LIN {X 0,Y 411.208,Z 237.264,A -85,B 0,C 180,E1 -10473.156,E2 -10473.156} C_VEL
LIN {X 0,Y 411.193,Z 237.263,A -85,B 0,C 180,E1 -10476.552,E2 -10476.552} C_VEL
LIN {X 0,Y 411.171,Z 237.27,A -85,B 0,C 180,E1 -10479.72,E2 -10479.72} C_VEL
LIN {X 0,Y 411.166,Z 237.272,A -85,B 0,C 180,E1 -10483.135,E2 -10483.135} C_VEL
LIN {X 0,Y 411.208,Z 237.375,A -85,B 0,C 180,E1 -10486.787,E2 -10486.787} C_VEL
LIN {X 0,Y 412.368,Z 243.528,A -85,B 0,C 180,E1 -10490.08,E2 -10490.08} C_VEL
LIN {X 0,Y 413.369,Z 249.555,A -85,B 0,C 180,E1 -10493.043,E2 -10493.043} C_VEL
LIN {X 0,Y 413.313,Z 254.436,A -85,B 0,C 180,E1 -10495.275,E2 -10495.275} C_VEL
LIN {X 0,Y 412.67,Z 262.638,A -85,B 0,C 180,E1 -10498.816,E2 -10498.816} C_VEL
LIN {X 0,Y 412.048,Z 271.447,A -85,B 0,C 180,E1 -10502.49,E2 -10502.49} C_VEL
LIN {X 0,Y 411.535,Z 279.596,A -85,B 0,C 180,E1 -10505.804,E2 -10505.804} C_VEL
LIN {X 0,Y 411.103,Z 287.435,A -85,B 0,C 180,E1 -10508.961,E2 -10508.961} C_VEL
LIN {X 0,Y 410.706,Z 295.977,A -85,B 0,C 180,E1 -10512.395,E2 -10512.395} C_VEL
LIN {X 0,Y 413.028,Z 310.701,A -85,B 0,C 180,E1 -10512.959,E2 -10512.959} C_VEL
LIN {X 0,Y 414.855,Z 323.572,A -85,B 0,C 180,E1 -10513.644,E2 -10513.644} C_VEL
LIN {X 0,Y 414.255,Z 335.281,A -85,B 0,C 180,E1 -10514.376,E2 -10514.376} C_VEL
LIN {X 0,Y 413.474,Z 345.991,A -85,B 0,C 180,E1 -10515.229,E2 -10515.229} C_VEL
LIN {X 0,Y 412.699,Z 356.944,A -85,B 0,C 180,E1 -10516.333,E2 -10516.333} C_VEL
LIN {X 0,Y 412.139,Z 365.888,A -85,B 0,C 180,E1 -10517.443,E2 -10517.443} C_VEL
LIN {X 0,Y 411.369,Z 375.605,A -85,B 0,C 180,E1 -10518.919,E2 -10518.919} C_VEL
LIN {X 0,Y 410.826,Z 383.351,A -85,B 0,C 180,E1 -10520.399,E2 -10520.399} C_VEL
LIN {X 0,Y 410.354,Z 390.497,A -85,B 0,C 180,E1 -10522.125,E2 -10522.125} C_VEL
LIN {X 0,Y 410.177,Z 395.261,A -85,B 0,C 180,E1 -10523.606,E2 -10523.606} C_VEL
LIN {X 0,Y 410.096,Z 398.905,A -85,B 0,C 180,E1 -10525.085,E2 -10525.085} C_VEL
LIN {X 0,Y 409.954,Z 400.778,A -85,B 0,C 180,E1 -10526.068,E2 -10526.068} C_VEL
LIN {X 0,Y 410.007,Z 402.193,A -85,B 0,C 180,E1 -10527.052,E2 -10527.052} C_VEL
LIN {X 0,Y 409.988,Z 403.2,A -85,B 0,C 180,E1 -10528.035,E2 -10528.035} C_VEL
LIN {X 0,Y 409.959,Z 403.813,A -85,B 0,C 180,E1 -10529.018,E2 -10529.018} C_VEL
LIN {X 0,Y 409.967,Z 404.032,A -85,B 0,C 180,E1 -10530,E2 -10530} C_VEL
LIN {X 0,Y 409.959,Z 403.813,A -85,B 0,C 180,E1 -10530.982,E2 -10530.982} C_VEL
LIN {X 0,Y 409.988,Z 403.201,A -85,B 0,C 180,E1 -10531.965,E2 -10531.965} C_VEL
LIN {X 0,Y 410.007,Z 402.196,A -85,B 0,C 180,E1 -10532.948,E2 -10532.948} C_VEL
LIN {X 0,Y 409.954,Z 400.782,A -85,B 0,C 180,E1 -10533.932,E2 -10533.932} C_VEL
LIN {X 0,Y 410.108,Z 397.823,A -85,B 0,C 180,E1 -10535.409,E2 -10535.409} C_VEL
LIN {X 0,Y 410.198,Z 393.812,A -85,B 0,C 180,E1 -10536.888,E2 -10536.888} C_VEL
LIN {X 0,Y 410.551,Z 387.657,A -85,B 0,C 180,E1 -10538.615,E2 -10538.615} C_VEL
LIN {X 0,Y 410.993,Z 380.936,A -85,B 0,C 180,E1 -10540.095,E2 -10540.095} C_VEL
LIN {X 0,Y 411.602,Z 372.606,A -85,B 0,C 180,E1 -10541.574,E2 -10541.574} C_VEL
LIN {X 0,Y 412.221,Z 364.073,A -85,B 0,C 180,E1 -10542.806,E2 -10542.806} C_VEL
LIN {X 0,Y 412.945,Z 354.501,A -85,B 0,C 180,E1 -10543.934,E2 -10543.934} C_VEL
LIN {X 0,Y 413.672,Z 343.125,A -85,B 0,C 180,E1 -10545.016,E2 -10545.016} C_VEL
LIN {X 0,Y 414.506,Z 331.727,A -85,B 0,C 180,E1 -10545.867,E2 -10545.867} C_VEL
LIN {X 0,Y 414.812,Z 323.512,A -85,B 0,C 180,E1 -10546.36,E2 -10546.36} C_VEL
LIN {X 0,Y 412.966,Z 310.197,A -85,B 0,C 180,E1 -10547.063,E2 -10547.063} C_VEL
LIN {X 0,Y 410.827,Z 297.222,A -85,B 0,C 180,E1 -10547.554,E2 -10547.554} C_VEL
LIN {X 0,Y 410.719,Z 295.854,A -85,B 0,C 180,E1 -10547.636,E2 -10547.636} C_VEL
LIN {X 0,Y 411.108,Z 287.427,A -85,B 0,C 180,E1 -10551.039,E2 -10551.039} C_VEL
LIN {X 0,Y 411.529,Z 279.586,A -85,B 0,C 180,E1 -10554.197,E2 -10554.197} C_VEL
LIN {X 0,Y 412.03,Z 271.406,A -85,B 0,C 180,E1 -10557.506,E2 -10557.506} C_VEL
LIN {X 0,Y 412.548,Z 263.641,A -85,B 0,C 180,E1 -10560.735,E2 -10560.735} C_VEL
LIN {X 0,Y 413.078,Z 257.152,A -85,B 0,C 180,E1 -10563.522,E2 -10563.522} C_VEL
LIN {X 0,Y 413.457,Z 251.781,A -85,B 0,C 180,E1 -10565.905,E2 -10565.905} C_VEL
LIN {X 0,Y 413.12,Z 247.857,A -85,B 0,C 180,E1 -10567.766,E2 -10567.766} C_VEL
LIN {X 0,Y 411.88,Z 240.822,A -85,B 0,C 180,E1 -10571.342,E2 -10571.342} C_VEL
LIN {X 0,Y 411.202,Z 237.271,A -85,B 0,C 180,E1 -10573.298,E2 -10573.298} C_VEL
LIN {X 0,Y 411.167,Z 237.271,A -85,B 0,C 180,E1 -10576.865,E2 -10576.865} C_VEL
LIN {X 0,Y 411.172,Z 237.267,A -85,B 0,C 180,E1 -10580.28,E2 -10580.28} C_VEL
LIN {X 0,Y 411.195,Z 237.263,A -85,B 0,C 180,E1 -10583.448,E2 -10583.448} C_VEL
LIN {X 0,Y 411.211,Z 237.264,A -85,B 0,C 180,E1 -10586.874,E2 -10586.874} C_VEL
LIN {X 0,Y 411.214,Z 237.264,A -85,B 0,C 180,E1 -10590.65,E2 -10590.65} C_VEL
LIN {X 0,Y 411.179,Z 237.264,A -85,B 0,C 180,E1 -10593.615,E2 -10593.615} C_VEL
LIN {X 0,Y 411.193,Z 237.263,A -85,B 0,C 180,E1 -10596.852,E2 -10596.852} C_VEL
LIN {X 0,Y 411.219,Z 237.264,A -85,B 0,C 180,E1 -10600.05,E2 -10600.05} C_VEL
LIN {X 0,Y 411.267,Z 237.254,A -85,B 0,C 180,E1 -10603.131,E2 -10603.131} C_VEL
LIN {X 0,Y 411.309,Z 237.248,A -85,B 0,C 180,E1 -10606.897,E2 -10606.897} C_VEL
LIN {X 0,Y 411.282,Z 237.254,A -85,B 0,C 180,E1 -10610.161,E2 -10610.161} C_VEL
LIN {X 0,Y 411.442,Z 237.233,A -85,B 0,C 180,E1 -10613.133,E2 -10613.133} C_VEL
LIN {X 0,Y 411.312,Z 237.25,A -85,B 0,C 180,E1 -10615.099,E2 -10615.099} C_VEL
LIN {X 0,Y 411.515,Z 237.224,A -85,B 0,C 180,E1 -10618.043,E2 -10618.043} C_VEL
LIN {X 0,Y 411.382,Z 237.241,A -85,B 0,C 180,E1 -10620.979,E2 -10620.979} C_VEL
LIN {X 0,Y 411.443,Z 237.233,A -85,B 0,C 180,E1 -10622.937,E2 -10622.937} C_VEL
LIN {X 0,Y 411.437,Z 237.233,A -85,B 0,C 180,E1 -10626.648,E2 -10626.648} C_VEL
LIN {X 0,Y 411.324,Z 237.25,A -85,B 0,C 180,E1 -10628.846,E2 -10628.846} C_VEL
LIN {X 0,Y 411.289,Z 237.252,A -85,B 0,C 180,E1 -10631.833,E2 -10631.833} C_VEL
LIN {X 0,Y 411.256,Z 237.258,A -85,B 0,C 180,E1 -10634.853,E2 -10634.853} C_VEL
LIN {X 0,Y 411.248,Z 237.255,A -85,B 0,C 180,E1 -10637.915,E2 -10637.915} C_VEL
LIN {X 0,Y 411.201,Z 237.265,A -85,B 0,C 180,E1 -10641.034,E2 -10641.034} C_VEL
LIN {X 0,Y 411.216,Z 237.262,A -85,B 0,C 180,E1 -10644.216,E2 -10644.216} C_VEL
LIN {X 0,Y 411.183,Z 237.264,A -85,B 0,C 180,E1 -10647.483,E2 -10647.483} C_VEL
LIN {X 0,Y 411.199,Z 237.262,A -85,B 0,C 180,E1 -10649.713,E2 -10649.713} C_VEL
LIN {X 0,Y 411.21,Z 237.261,A -85,B 0,C 180,E1 -10653.156,E2 -10653.156} C_VEL
LIN {X 0,Y 411.196,Z 237.266,A -85,B 0,C 180,E1 -10656.552,E2 -10656.552} C_VEL
LIN {X 0,Y 411.21,Z 237.263,A -85,B 0,C 180,E1 -10659.727,E2 -10659.727} C_VEL
LIN {X 0,Y 411.174,Z 237.265,A -85,B 0,C 180,E1 -10663.134,E2 -10663.134} C_VEL
LIN {X 0,Y 411.171,Z 237.269,A -85,B 0,C 180,E1 -10665.881,E2 -10665.881} C_VEL
LIN {X 0,Y 411.163,Z 237.267,A -85,B 0,C 180,E1 -10668.772,E2 -10668.772} C_VEL
LIN {X 0,Y 411.191,Z 237.267,A -85,B 0,C 180,E1 -10672.025,E2 -10672.025} C_VEL
LIN {X 0,Y 411.078,Z 237.279,A -85,B 0,C 180,E1 -10675.149,E2 -10675.149} C_VEL
LIN {X 0,Y 410.719,Z 237.327,A -85,B 0,C 180,E1 -10677.963,E2 -10677.963} C_VEL
LIN {X 0,Y 410.617,Z 239.167,A -85,B 0,C 180,E1 -10680.24,E2 -10680.24} C_VEL
LIN {X 0,Y 410.512,Z 242.3,A -85,B 0,C 180,E1 -10683.569,E2 -10683.569} C_VEL
LIN {X 0,Y 410.497,Z 244.4,A -85,B 0,C 180,E1 -10685.738,E2 -10685.738} C_VEL
LIN {X 0,Y 410.419,Z 247.648,A -85,B 0,C 180,E1 -10688.924,E2 -10688.924} C_VEL
LIN {X 0,Y 410.4,Z 251.592,A -85,B 0,C 180,E1 -10692.501,E2 -10692.501} C_VEL
LIN {X 0,Y 414.208,Z 265.973,A -85,B 0,C 180,E1 -10693.18,E2 -10693.18} C_VEL
LIN {X 0,Y 415.689,Z 273.997,A -85,B 0,C 180,E1 -10693.638,E2 -10693.638} C_VEL
LIN {X 0,Y 415.064,Z 286.501,A -85,B 0,C 180,E1 -10694.407,E2 -10694.407} C_VEL
LIN {X 0,Y 414.427,Z 297.234,A -85,B 0,C 180,E1 -10695.263,E2 -10695.263} C_VEL
LIN {X 0,Y 413.779,Z 307.095,A -85,B 0,C 180,E1 -10696.244,E2 -10696.244} C_VEL
LIN {X 0,Y 412.992,Z 317.038,A -85,B 0,C 180,E1 -10697.469,E2 -10697.469} C_VEL
LIN {X 0,Y 412.244,Z 326.64,A -85,B 0,C 180,E1 -10698.942,E2 -10698.942} C_VEL
LIN {X 0,Y 411.583,Z 334.299,A -85,B 0,C 180,E1 -10700.416,E2 -10700.416} C_VEL
LIN {X 0,Y 411.025,Z 341.318,A -85,B 0,C 180,E1 -10702.138,E2 -10702.138} C_VEL
LIN {X 0,Y 410.699,Z 345.99,A -85,B 0,C 180,E1 -10703.614,E2 -10703.614} C_VEL
LIN {X 0,Y 410.418,Z 349.569,A -85,B 0,C 180,E1 -10705.088,E2 -10705.088} C_VEL
LIN {X 0,Y 410.412,Z 351.41,A -85,B 0,C 180,E1 -10706.072,E2 -10706.072} C_VEL
LIN {X 0,Y 410.276,Z 352.804,A -85,B 0,C 180,E1 -10707.054,E2 -10707.054} C_VEL
LIN {X 0,Y 410.078,Z 354.408,A -85,B 0,C 180,E1 -10709.018,E2 -10709.018} C_VEL
LIN {X 0,Y 410.074,Z 354.64,A -85,B 0,C 180,E1 -10710,E2 -10710} C_VEL
LIN {X 0,Y 410.139,Z 353.873,A -85,B 0,C 180,E1 -10711.964,E2 -10711.964} C_VEL
LIN {X 0,Y 410.408,Z 351.56,A -85,B 0,C 180,E1 -10713.928,E2 -10713.928} C_VEL
LIN {X 0,Y 410.42,Z 348.726,A -85,B 0,C 180,E1 -10715.404,E2 -10715.404} C_VEL
LIN {X 0,Y 410.796,Z 344.12,A -85,B 0,C 180,E1 -10717.123,E2 -10717.123} C_VEL
LIN {X 0,Y 411.267,Z 337.92,A -85,B 0,C 180,E1 -10718.847,E2 -10718.847} C_VEL
LIN {X 0,Y 411.417,Z 336.229,A -85,B 0,C 180,E1 -10719.249,E2 -10719.249} C_VEL
LIN {X 0,Y 411.057,Z 333.143,A -85,B 0,C 180,E1 -10719.946,E2 -10719.946} C_VEL
LIN {X 0,Y 407.66,Z 325.609,A -85,B 0,C 180,E1 -10721.511,E2 -10721.511} C_VEL
LIN {X 0,Y 406.164,Z 320.726,A -85,B 0,C 180,E1 -10722.362,E2 -10722.362} C_VEL
LIN {X 0,Y 406.065,Z 318.007,A -85,B 0,C 180,E1 -10722.768,E2 -10722.768} C_VEL
LIN {X 0,Y 406.893,Z 308.344,A -85,B 0,C 180,E1 -10723.994,E2 -10723.994} C_VEL
LIN {X 0,Y 407.587,Z 297.853,A -85,B 0,C 180,E1 -10725.07,E2 -10725.07} C_VEL
LIN {X 0,Y 408.319,Z 286.508,A -85,B 0,C 180,E1 -10725.985,E2 -10725.985} C_VEL
LIN {X 0,Y 408.902,Z 274.466,A -85,B 0,C 180,E1 -10726.737,E2 -10726.737} C_VEL
LIN {X 0,Y 406.265,Z 262.744,A -85,B 0,C 180,E1 -10727.417,E2 -10727.417} C_VEL
LIN {X 0,Y 403.333,Z 251.921,A -85,B 0,C 180,E1 -10727.934,E2 -10727.934} C_VEL
LIN {X 0,Y 403.334,Z 249.256,A -85,B 0,C 180,E1 -10730.395,E2 -10730.395} C_VEL
LIN {X 0,Y 403.403,Z 245.95,A -85,B 0,C 180,E1 -10733.622,E2 -10733.622} C_VEL
LIN {X 0,Y 403.481,Z 242.745,A -85,B 0,C 180,E1 -10736.929,E2 -10736.929} C_VEL
LIN {X 0,Y 403.612,Z 239.579,A -85,B 0,C 180,E1 -10740.329,E2 -10740.329} C_VEL
LIN {X 0,Y 403.631,Z 238.502,A -85,B 0,C 180,E1 -10741.491,E2 -10741.491} C_VEL
LIN {X 0,Y 403.873,Z 238.178,A -85,B 0,C 180,E1 -10743.838,E2 -10743.838} C_VEL
LIN {X 0,Y 404.097,Z 238.151,A -85,B 0,C 180,E1 -10746.251,E2 -10746.251} C_VEL
LIN {X 0,Y 404.15,Z 238.141,A -85,B 0,C 180,E1 -10748.758,E2 -10748.758} C_VEL
LIN {X 0,Y 404.121,Z 238.145,A -85,B 0,C 180,E1 -10751.599,E2 -10751.599} C_VEL
LIN {X 0,Y 404.147,Z 238.141,A -85,B 0,C 180,E1 -10754.522,E2 -10754.522} C_VEL
LIN {X 0,Y 404.134,Z 238.143,A -85,B 0,C 180,E1 -10757.295,E2 -10757.295} C_VEL
LIN {X 0,Y 404.171,Z 238.142,A -85,B 0,C 180,E1 -10759.955,E2 -10759.955} C_VEL
LIN {X 0,Y 404.137,Z 238.143,A -85,B 0,C 180,E1 -10763.125,E2 -10763.125} C_VEL
LIN {X 0,Y 404.147,Z 238.141,A -85,B 0,C 180,E1 -10766.188,E2 -10766.188} C_VEL
LIN {X 0,Y 404.146,Z 238.144,A -85,B 0,C 180,E1 -10769.715,E2 -10769.715} C_VEL
LIN {X 0,Y 404.131,Z 238.146,A -85,B 0,C 180,E1 -10773.118,E2 -10773.118} C_VEL
LIN {X 0,Y 404.163,Z 238.139,A -85,B 0,C 180,E1 -10776.425,E2 -10776.425} C_VEL
LIN {X 0,Y 404.194,Z 238.135,A -85,B 0,C 180,E1 -10779.874,E2 -10779.874} C_VEL
LIN {X 0,Y 404.218,Z 238.136,A -85,B 0,C 180,E1 -10782.993,E2 -10782.993} C_VEL
LIN {X 0,Y 404.285,Z 238.128,A -85,B 0,C 180,E1 -10786.939,E2 -10786.939} C_VEL
LIN {X 0,Y 404.261,Z 238.126,A -85,B 0,C 180,E1 -10789.988,E2 -10789.988} C_VEL
LIN {X 0,Y 404.413,Z 238.112,A -85,B 0,C 180,E1 -10793.013,E2 -10793.013} C_VEL
LIN {X 0,Y 404.277,Z 238.127,A -85,B 0,C 180,E1 -10795.013,E2 -10795.013} C_VEL
LIN {X 0,Y 404.477,Z 238.099,A -85,B 0,C 180,E1 -10798.008,E2 -10798.008} C_VEL
LIN {X 0,Y 404.412,Z 238.109,A -85,B 0,C 180,E1 -10800.996,E2 -10800.996} C_VEL
LIN {X 0,Y 404.418,Z 238.108,A -85,B 0,C 180,E1 -10802.988,E2 -10802.988} C_VEL
LIN {X 0,Y 404.417,Z 238.109,A -85,B 0,C 180,E1 -10805.985,E2 -10805.985} C_VEL
LIN {X 0,Y 404.265,Z 238.126,A -85,B 0,C 180,E1 -10809.002,E2 -10809.002} C_VEL
LIN {X 0,Y 404.252,Z 238.131,A -85,B 0,C 180,E1 -10812.042,E2 -10812.042} C_VEL
LIN {X 0,Y 404.207,Z 238.133,A -85,B 0,C 180,E1 -10815.118,E2 -10815.118} C_VEL
LIN {X 0,Y 404.213,Z 238.136,A -85,B 0,C 180,E1 -10818.238,E2 -10818.238} C_VEL
LIN {X 0,Y 404.141,Z 238.143,A -85,B 0,C 180,E1 -10821.419,E2 -10821.419} C_VEL
LIN {X 0,Y 404.15,Z 238.139,A -85,B 0,C 180,E1 -10824.667,E2 -10824.667} C_VEL
LIN {X 0,Y 404.117,Z 238.147,A -85,B 0,C 180,E1 -10828.006,E2 -10828.006} C_VEL
LIN {X 0,Y 404.145,Z 238.141,A -85,B 0,C 180,E1 -10830.285,E2 -10830.285} C_VEL
LIN {X 0,Y 404.147,Z 238.144,A -85,B 0,C 180,E1 -10833.812,E2 -10833.812} C_VEL
LIN {X 0,Y 404.136,Z 238.143,A -85,B 0,C 180,E1 -10836.875,E2 -10836.875} C_VEL
LIN {X 0,Y 404.118,Z 238.148,A -85,B 0,C 180,E1 -10840.075,E2 -10840.075} C_VEL
LIN {X 0,Y 404.146,Z 238.146,A -85,B 0,C 180,E1 -10843.082,E2 -10843.082} C_VEL
LIN {X 0,Y 404.134,Z 238.19,A -85,B 0,C 180,E1 -10846.377,E2 -10846.377} C_VEL
LIN {X 0,Y 405.31,Z 244.339,A -85,B 0,C 180,E1 -10849.725,E2 -10849.725} C_VEL
LIN {X 0,Y 406.3,Z 250.268,A -85,B 0,C 180,E1 -10852.741,E2 -10852.741} C_VEL
LIN {X 0,Y 406.439,Z 253.688,A -85,B 0,C 180,E1 -10854.362,E2 -10854.362} C_VEL
LIN {X 0,Y 405.883,Z 260.785,A -85,B 0,C 180,E1 -10857.535,E2 -10857.535} C_VEL
LIN {X 0,Y 405.192,Z 270.028,A -85,B 0,C 180,E1 -10861.511,E2 -10861.511} C_VEL
LIN {X 0,Y 404.645,Z 277.382,A -85,B 0,C 180,E1 -10864.576,E2 -10864.576} C_VEL
LIN {X 0,Y 404.164,Z 285.773,A -85,B 0,C 180,E1 -10868.046,E2 -10868.046} C_VEL
LIN {X 0,Y 403.76,Z 293.477,A -85,B 0,C 180,E1 -10871.215,E2 -10871.215} C_VEL
LIN {X 0,Y 403.657,Z 295.615,A -85,B 0,C 180,E1 -10872.096,E2 -10872.096} C_VEL
LIN {X 0,Y 405.857,Z 309.059,A -85,B 0,C 180,E1 -10872.599,E2 -10872.599} C_VEL
LIN {X 0,Y 407.618,Z 321.66,A -85,B 0,C 180,E1 -10873.262,E2 -10873.262} C_VEL
LIN {X 0,Y 407.968,Z 325.895,A -85,B 0,C 180,E1 -10873.519,E2 -10873.519} C_VEL
LIN {X 0,Y 407.146,Z 338.138,A -85,B 0,C 180,E1 -10874.353,E2 -10874.353} C_VEL
LIN {X 0,Y 406.275,Z 349.873,A -85,B 0,C 180,E1 -10875.384,E2 -10875.384} C_VEL
LIN {X 0,Y 405.538,Z 359.806,A -85,B 0,C 180,E1 -10876.481,E2 -10876.481} C_VEL
LIN {X 0,Y 404.876,Z 368.943,A -85,B 0,C 180,E1 -10877.723,E2 -10877.723} C_VEL
LIN {X 0,Y 404.106,Z 377.929,A -85,B 0,C 180,E1 -10879.225,E2 -10879.225} C_VEL
LIN {X 0,Y 403.612,Z 385.174,A -85,B 0,C 180,E1 -10880.731,E2 -10880.731} C_VEL
LIN {X 0,Y 403.301,Z 390.068,A -85,B 0,C 180,E1 -10881.986,E2 -10881.986} C_VEL
LIN {X 0,Y 403.104,Z 395.159,A -85,B 0,C 180,E1 -10883.607,E2 -10883.607} C_VEL
LIN {X 0,Y 403.008,Z 398.476,A -85,B 0,C 180,E1 -10884.998,E2 -10884.998} C_VEL
LIN {X 0,Y 402.877,Z 400.351,A -85,B 0,C 180,E1 -10885.999,E2 -10885.999} C_VEL
LIN {X 0,Y 402.909,Z 401.765,A -85,B 0,C 180,E1 -10887,E2 -10887} C_VEL
LIN {X 0,Y 402.921,Z 402.774,A -85,B 0,C 180,E1 -10888.001,E2 -10888.001} C_VEL
LIN {X 0,Y 402.884,Z 403.387,A -85,B 0,C 180,E1 -10889.001,E2 -10889.001} C_VEL
LIN {X 0,Y 402.89,Z 403.606,A -85,B 0,C 180,E1 -10890,E2 -10890} C_VEL
LIN {X 0,Y 402.884,Z 403.387,A -85,B 0,C 180,E1 -10891,E2 -10891} C_VEL
LIN {X 0,Y 402.921,Z 402.775,A -85,B 0,C 180,E1 -10891.999,E2 -10891.999} C_VEL
LIN {X 0,Y 402.909,Z 401.768,A -85,B 0,C 180,E1 -10893,E2 -10893} C_VEL
LIN {X 0,Y 402.877,Z 400.354,A -85,B 0,C 180,E1 -10894.001,E2 -10894.001} C_VEL
LIN {X 0,Y 403.006,Z 397.393,A -85,B 0,C 180,E1 -10895.504,E2 -10895.504} C_VEL
LIN {X 0,Y 403.117,Z 393.382,A -85,B 0,C 180,E1 -10897.01,E2 -10897.01} C_VEL
LIN {X 0,Y 403.517,Z 387.227,A -85,B 0,C 180,E1 -10898.766,E2 -10898.766} C_VEL
LIN {X 0,Y 403.966,Z 380.505,A -85,B 0,C 180,E1 -10900.272,E2 -10900.272} C_VEL
LIN {X 0,Y 404.609,Z 372.175,A -85,B 0,C 180,E1 -10901.777,E2 -10901.777} C_VEL
LIN {X 0,Y 405.239,Z 363.64,A -85,B 0,C 180,E1 -10903.03,E2 -10903.03} C_VEL
LIN {X 0,Y 406.02,Z 353.608,A -85,B 0,C 180,E1 -10904.226,E2 -10904.226} C_VEL
LIN {X 0,Y 406.791,Z 342.693,A -85,B 0,C 180,E1 -10905.276,E2 -10905.276} C_VEL
LIN {X 0,Y 407.668,Z 331.405,A -85,B 0,C 180,E1 -10906.132,E2 -10906.132} C_VEL
LIN {X 0,Y 407.869,Z 323.777,A -85,B 0,C 180,E1 -10906.606,E2 -10906.606} C_VEL
LIN {X 0,Y 406.095,Z 310.832,A -85,B 0,C 180,E1 -10907.316,E2 -10907.316} C_VEL
LIN {X 0,Y 403.909,Z 297.405,A -85,B 0,C 180,E1 -10907.851,E2 -10907.851} C_VEL
LIN {X 0,Y 403.657,Z 295.556,A -85,B 0,C 180,E1 -10907.904,E2 -10907.904} C_VEL
LIN {X 0,Y 404.099,Z 287.058,A -85,B 0,C 180,E1 -10911.422,E2 -10911.422} C_VEL
LIN {X 0,Y 404.528,Z 279.25,A -85,B 0,C 180,E1 -10914.643,E2 -10914.643} C_VEL
LIN {X 0,Y 405.09,Z 271.299,A -85,B 0,C 180,E1 -10917.933,E2 -10917.933} C_VEL
LIN {X 0,Y 405.818,Z 261.933,A -85,B 0,C 180,E1 -10921.941,E2 -10921.941} C_VEL
LIN {X 0,Y 406.33,Z 255.462,A -85,B 0,C 180,E1 -10924.805,E2 -10924.805} C_VEL
LIN {X 0,Y 406.444,Z 251.552,A -85,B 0,C 180,E1 -10926.624,E2 -10926.624} C_VEL
LIN {X 0,Y 405.629,Z 246.233,A -85,B 0,C 180,E1 -10929.288,E2 -10929.288} C_VEL
LIN {X 0,Y 404.5,Z 239.906,A -85,B 0,C 180,E1 -10932.657,E2 -10932.657} C_VEL
LIN {X 0,Y 404.135,Z 238.15,A -85,B 0,C 180,E1 -10933.673,E2 -10933.673} C_VEL
LIN {X 0,Y 404.147,Z 238.146,A -85,B 0,C 180,E1 -10936.918,E2 -10936.918} C_VEL
LIN {X 0,Y 404.135,Z 238.141,A -85,B 0,C 180,E1 -10939.951,E2 -10939.951} C_VEL
LIN {X 0,Y 404.138,Z 238.143,A -85,B 0,C 180,E1 -10943.126,E2 -10943.126} C_VEL
LIN {X 0,Y 404.148,Z 238.144,A -85,B 0,C 180,E1 -10946.188,E2 -10946.188} C_VEL
LIN {X 0,Y 404.147,Z 238.141,A -85,B 0,C 180,E1 -10949.715,E2 -10949.715} C_VEL
LIN {X 0,Y 404.122,Z 238.143,A -85,B 0,C 180,E1 -10953.118,E2 -10953.118} C_VEL
LIN {X 0,Y 404.153,Z 238.143,A -85,B 0,C 180,E1 -10956.424,E2 -10956.424} C_VEL
LIN {X 0,Y 404.195,Z 238.139,A -85,B 0,C 180,E1 -10959.874,E2 -10959.874} C_VEL
LIN {X 0,Y 404.22,Z 238.131,A -85,B 0,C 180,E1 -10962.993,E2 -10962.993} C_VEL
LIN {X 0,Y 404.287,Z 238.122,A -85,B 0,C 180,E1 -10966.939,E2 -10966.939} C_VEL
LIN {X 0,Y 404.249,Z 238.131,A -85,B 0,C 180,E1 -10969.988,E2 -10969.988} C_VEL
LIN {X 0,Y 404.391,Z 238.111,A -85,B 0,C 180,E1 -10973.012,E2 -10973.012} C_VEL
LIN {X 0,Y 404.284,Z 238.125,A -85,B 0,C 180,E1 -10975.014,E2 -10975.014} C_VEL
LIN {X 0,Y 404.484,Z 238.1,A -85,B 0,C 180,E1 -10978.009,E2 -10978.009} C_VEL
LIN {X 0,Y 404.352,Z 238.117,A -85,B 0,C 180,E1 -10980.996,E2 -10980.996} C_VEL
LIN {X 0,Y 404.402,Z 238.11,A -85,B 0,C 180,E1 -10982.989,E2 -10982.989} C_VEL
LIN {X 0,Y 404.385,Z 238.112,A -85,B 0,C 180,E1 -10986.647,E2 -10986.647} C_VEL
LIN {X 0,Y 404.262,Z 238.126,A -85,B 0,C 180,E1 -10990.012,E2 -10990.012} C_VEL
LIN {X 0,Y 404.271,Z 238.13,A -85,B 0,C 180,E1 -10993.211,E2 -10993.211} C_VEL
LIN {X 0,Y 404.22,Z 238.136,A -85,B 0,C 180,E1 -10997.007,E2 -10997.007} C_VEL
LIN {X 0,Y 404.168,Z 238.139,A -85,B 0,C 180,E1 -11000.351,E2 -11000.351} C_VEL
LIN {X 0,Y 404.165,Z 238.138,A -85,B 0,C 180,E1 -11003.575,E2 -11003.575} C_VEL
LIN {X 0,Y 404.133,Z 238.146,A -85,B 0,C 180,E1 -11006.882,E2 -11006.882} C_VEL
LIN {X 0,Y 404.146,Z 238.144,A -85,B 0,C 180,E1 -11010.285,E2 -11010.285} C_VEL
LIN {X 0,Y 404.148,Z 238.141,A -85,B 0,C 180,E1 -11013.812,E2 -11013.812} C_VEL
LIN {X 0,Y 404.139,Z 238.143,A -85,B 0,C 180,E1 -11016.875,E2 -11016.875} C_VEL
LIN {X 0,Y 404.151,Z 238.144,A -85,B 0,C 180,E1 -11020.08,E2 -11020.08} C_VEL
LIN {X 0,Y 404.154,Z 238.139,A -85,B 0,C 180,E1 -11023.083,E2 -11023.083} C_VEL
LIN {X 0,Y 404.151,Z 238.144,A -85,B 0,C 180,E1 -11025.926,E2 -11025.926} C_VEL
LIN {X 0,Y 404.118,Z 238.145,A -85,B 0,C 180,E1 -11028.634,E2 -11028.634} C_VEL
LIN {X 0,Y 404.15,Z 238.143,A -85,B 0,C 180,E1 -11031.493,E2 -11031.493} C_VEL
LIN {X 0,Y 404.043,Z 238.153,A -85,B 0,C 180,E1 -11034.838,E2 -11034.838} C_VEL
LIN {X 0,Y 403.728,Z 238.197,A -85,B 0,C 180,E1 -11037.34,E2 -11037.34} C_VEL
LIN {X 0,Y 403.618,Z 238.475,A -85,B 0,C 180,E1 -11038.563,E2 -11038.563} C_VEL
LIN {X 0,Y 403.6,Z 240.522,A -85,B 0,C 180,E1 -11040.819,E2 -11040.819} C_VEL
LIN {X 0,Y 403.459,Z 243.691,A -85,B 0,C 180,E1 -11044.184,E2 -11044.184} C_VEL
LIN {X 0,Y 403.384,Z 246.932,A -85,B 0,C 180,E1 -11047.462,E2 -11047.462} C_VEL
LIN {X 0,Y 403.368,Z 250.306,A -85,B 0,C 180,E1 -11050.668,E2 -11050.668} C_VEL
LIN {X 0,Y 403.337,Z 251.989,A -85,B 0,C 180,E1 -11052.19,E2 -11052.19} C_VEL
LIN {X 0,Y 407.009,Z 265.767,A -85,B 0,C 180,E1 -11052.845,E2 -11052.845} C_VEL
LIN {X 0,Y 408.821,Z 273.82,A -85,B 0,C 180,E1 -11053.32,E2 -11053.32} C_VEL
LIN {X 0,Y 408.332,Z 285.176,A -85,B 0,C 180,E1 -11054.015,E2 -11054.015} C_VEL
LIN {X 0,Y 407.742,Z 295.816,A -85,B 0,C 180,E1 -11054.849,E2 -11054.849} C_VEL
LIN {X 0,Y 406.991,Z 306.505,A -85,B 0,C 180,E1 -11055.897,E2 -11055.897} C_VEL
LIN {X 0,Y 406.229,Z 315.664,A -85,B 0,C 180,E1 -11057.002,E2 -11057.002} C_VEL
LIN {X 0,Y 405.543,Z 324.126,A -85,B 0,C 180,E1 -11058.251,E2 -11058.251} C_VEL
LIN {X 0,Y 404.85,Z 332.34,A -85,B 0,C 180,E1 -11059.75,E2 -11059.75} C_VEL
LIN {X 0,Y 404.294,Z 337.962,A -85,B 0,C 180,E1 -11060.999,E2 -11060.999} C_VEL
LIN {X 0,Y 403.806,Z 344.299,A -85,B 0,C 180,E1 -11062.773,E2 -11062.773} C_VEL
LIN {X 0,Y 403.386,Z 348.945,A -85,B 0,C 180,E1 -11064.501,E2 -11064.501} C_VEL
LIN {X 0,Y 403.357,Z 351.836,A -85,B 0,C 180,E1 -11066.003,E2 -11066.003} C_VEL
LIN {X 0,Y 403.215,Z 353.23,A -85,B 0,C 180,E1 -11067.002,E2 -11067.002} C_VEL
LIN {X 0,Y 402.999,Z 354.835,A -85,B 0,C 180,E1 -11069.001,E2 -11069.001} C_VEL
LIN {X 0,Y 402.992,Z 355.067,A -85,B 0,C 180,E1 -11070,E2 -11070} C_VEL
LIN {X 0,Y 403.068,Z 354.298,A -85,B 0,C 180,E1 -11071.998,E2 -11071.998} C_VEL
LIN {X 0,Y 403.353,Z 351.986,A -85,B 0,C 180,E1 -11073.996,E2 -11073.996} C_VEL
LIN {X 0,Y 403.366,Z 349.151,A -85,B 0,C 180,E1 -11075.499,E2 -11075.499} C_VEL
LIN {X 0,Y 403.758,Z 344.778,A -85,B 0,C 180,E1 -11077.174,E2 -11077.174} C_VEL
LIN {X 0,Y 404.096,Z 340.306,A -85,B 0,C 180,E1 -11078.501,E2 -11078.501} C_VEL
LIN {X 0,Y 404.687,Z 334.026,A -85,B 0,C 180,E1 -11080.001,E2 -11080.001} C_VEL
LIN {X 0,Y 405.357,Z 326.163,A -85,B 0,C 180,E1 -11081.501,E2 -11081.501} C_VEL
LIN {X 0,Y 406.065,Z 318.007,A -85,B 0,C 180,E1 -11082.768,E2 -11082.768} C_VEL
LIN {X 0,Y 405.738,Z 313.854,A -85,B 0,C 180,E1 -11083.357,E2 -11083.357} C_VEL
LIN {X 0,Y 403.51,Z 306.894,A -85,B 0,C 180,E1 -11084.306,E2 -11084.306} C_VEL
LIN {X 0,Y 401.317,Z 299.494,A -85,B 0,C 180,E1 -11085.188,E2 -11085.188} C_VEL
LIN {X 0,Y 401.034,Z 294.563,A -85,B 0,C 180,E1 -11085.662,E2 -11085.662} C_VEL
LIN {X 0,Y 401.716,Z 283.952,A -85,B 0,C 180,E1 -11086.475,E2 -11086.475} C_VEL
LIN {X 0,Y 402.093,Z 275.613,A -85,B 0,C 180,E1 -11086.986,E2 -11086.986} C_VEL
LIN {X 0,Y 399.407,Z 263.783,A -85,B 0,C 180,E1 -11087.699,E2 -11087.699} C_VEL
LIN {X 0,Y 396.282,Z 252.362,A -85,B 0,C 180,E1 -11088.243,E2 -11088.243} C_VEL
LIN {X 0,Y 396.29,Z 249.653,A -85,B 0,C 180,E1 -11090.774,E2 -11090.774} C_VEL
LIN {X 0,Y 396.376,Z 246.326,A -85,B 0,C 180,E1 -11094.067,E2 -11094.067} C_VEL
LIN {X 0,Y 396.444,Z 242.973,A -85,B 0,C 180,E1 -11097.578,E2 -11097.578} C_VEL
LIN {X 0,Y 396.569,Z 239.883,A -85,B 0,C 180,E1 -11100.927,E2 -11100.927} C_VEL
LIN {X 0,Y 396.604,Z 239.085,A -85,B 0,C 180,E1 -11102.115,E2 -11102.115} C_VEL
LIN {X 0,Y 396.914,Z 239.046,A -85,B 0,C 180,E1 -11104.514,E2 -11104.514} C_VEL
LIN {X 0,Y 397.081,Z 239.02,A -85,B 0,C 180,E1 -11107.206,E2 -11107.206} C_VEL
LIN {X 0,Y 397.103,Z 239.021,A -85,B 0,C 180,E1 -11110.445,E2 -11110.445} C_VEL
LIN {X 0,Y 397.102,Z 239.02,A -85,B 0,C 180,E1 -11113.649,E2 -11113.649} C_VEL
LIN {X 0,Y 397.103,Z 239.019,A -85,B 0,C 180,E1 -11116.521,E2 -11116.521} C_VEL
LIN {X 0,Y 397.114,Z 239.017,A -85,B 0,C 180,E1 -11120.423,E2 -11120.423} C_VEL
LIN {X 0,Y 397.11,Z 239.018,A -85,B 0,C 180,E1 -11124.265,E2 -11124.265} C_VEL
LIN {X 0,Y 397.116,Z 239.016,A -85,B 0,C 180,E1 -11126.727,E2 -11126.727} C_VEL
LIN {X 0,Y 397.119,Z 239.015,A -85,B 0,C 180,E1 -11130.295,E2 -11130.295} C_VEL
LIN {X 0,Y 397.093,Z 239.022,A -85,B 0,C 180,E1 -11133.739,E2 -11133.739} C_VEL
LIN {X 0,Y 397.107,Z 239.022,A -85,B 0,C 180,E1 -11137.085,E2 -11137.085} C_VEL
LIN {X 0,Y 397.149,Z 239.012,A -85,B 0,C 180,E1 -11140.353,E2 -11140.353} C_VEL
LIN {X 0,Y 397.166,Z 239.011,A -85,B 0,C 180,E1 -11143.553,E2 -11143.553} C_VEL
LIN {X 0,Y 397.231,Z 239.005,A -85,B 0,C 180,E1 -11146.703,E2 -11146.703} C_VEL
LIN {X 0,Y 397.221,Z 239.003,A -85,B 0,C 180,E1 -11149.809,E2 -11149.809} C_VEL
LIN {X 0,Y 397.365,Z 238.99,A -85,B 0,C 180,E1 -11152.888,E2 -11152.888} C_VEL
LIN {X 0,Y 397.25,Z 239.003,A -85,B 0,C 180,E1 -11154.925,E2 -11154.925} C_VEL
LIN {X 0,Y 397.446,Z 238.975,A -85,B 0,C 180,E1 -11157.973,E2 -11157.973} C_VEL
LIN {X 0,Y 397.377,Z 238.985,A -85,B 0,C 180,E1 -11161.013,E2 -11161.013} C_VEL
LIN {X 0,Y 397.377,Z 238.985,A -85,B 0,C 180,E1 -11163.041,E2 -11163.041} C_VEL
LIN {X 0,Y 397.367,Z 238.988,A -85,B 0,C 180,E1 -11166.092,E2 -11166.092} C_VEL
LIN {X 0,Y 397.235,Z 239.001,A -85,B 0,C 180,E1 -11169.162,E2 -11169.162} C_VEL
LIN {X 0,Y 397.217,Z 239.008,A -85,B 0,C 180,E1 -11172.258,E2 -11172.258} C_VEL
LIN {X 0,Y 397.18,Z 239.008,A -85,B 0,C 180,E1 -11175.392,E2 -11175.392} C_VEL
LIN {X 0,Y 397.165,Z 239.011,A -85,B 0,C 180,E1 -11178.573,E2 -11178.573} C_VEL
LIN {X 0,Y 397.097,Z 239.023,A -85,B 0,C 180,E1 -11181.819,E2 -11181.819} C_VEL
LIN {X 0,Y 397.098,Z 239.019,A -85,B 0,C 180,E1 -11185.136,E2 -11185.136} C_VEL
LIN {X 0,Y 397.071,Z 239.021,A -85,B 0,C 180,E1 -11188.548,E2 -11188.548} C_VEL
LIN {X 0,Y 397.084,Z 239.024,A -85,B 0,C 180,E1 -11191.836,E2 -11191.836} C_VEL
LIN {X 0,Y 397.127,Z 239.015,A -85,B 0,C 180,E1 -11194.493,E2 -11194.493} C_VEL
LIN {X 0,Y 397.093,Z 239.018,A -85,B 0,C 180,E1 -11198.276,E2 -11198.276} C_VEL
LIN {X 0,Y 397.055,Z 239.026,A -85,B 0,C 180,E1 -11201.977,E2 -11201.977} C_VEL
LIN {X 0,Y 397.088,Z 239.021,A -85,B 0,C 180,E1 -11205.069,E2 -11205.069} C_VEL
LIN {X 0,Y 397.128,Z 239.171,A -85,B 0,C 180,E1 -11206.048,E2 -11206.048} C_VEL
LIN {X 0,Y 398.248,Z 245.112,A -85,B 0,C 180,E1 -11209.362,E2 -11209.362} C_VEL
LIN {X 0,Y 399.25,Z 250.89,A -85,B 0,C 180,E1 -11212.386,E2 -11212.386} C_VEL
LIN {X 0,Y 399.429,Z 255.273,A -85,B 0,C 180,E1 -11214.504,E2 -11214.504} C_VEL
LIN {X 0,Y 398.781,Z 263.162,A -85,B 0,C 180,E1 -11218.082,E2 -11218.082} C_VEL
LIN {X 0,Y 398.073,Z 272.07,A -85,B 0,C 180,E1 -11221.976,E2 -11221.976} C_VEL
LIN {X 0,Y 397.459,Z 280.227,A -85,B 0,C 180,E1 -11225.447,E2 -11225.447} C_VEL
LIN {X 0,Y 396.935,Z 289.268,A -85,B 0,C 180,E1 -11229.261,E2 -11229.261} C_VEL
LIN {X 0,Y 396.609,Z 295.209,A -85,B 0,C 180,E1 -11231.768,E2 -11231.768} C_VEL
LIN {X 0,Y 398.856,Z 308.766,A -85,B 0,C 180,E1 -11232.289,E2 -11232.289} C_VEL
LIN {X 0,Y 400.519,Z 320.916,A -85,B 0,C 180,E1 -11232.939,E2 -11232.939} C_VEL
LIN {X 0,Y 401.106,Z 325.883,A -85,B 0,C 180,E1 -11233.256,E2 -11233.256} C_VEL
LIN {X 0,Y 400.284,Z 337.712,A -85,B 0,C 180,E1 -11234.078,E2 -11234.078} C_VEL
LIN {X 0,Y 399.379,Z 349.446,A -85,B 0,C 180,E1 -11235.126,E2 -11235.126} C_VEL
LIN {X 0,Y 398.561,Z 359.8,A -85,B 0,C 180,E1 -11236.295,E2 -11236.295} C_VEL
LIN {X 0,Y 397.915,Z 368.516,A -85,B 0,C 180,E1 -11237.505,E2 -11237.505} C_VEL
LIN {X 0,Y 397.097,Z 377.501,A -85,B 0,C 180,E1 -11239.032,E2 -11239.032} C_VEL
LIN {X 0,Y 396.569,Z 384.746,A -85,B 0,C 180,E1 -11240.565,E2 -11240.565} C_VEL
LIN {X 0,Y 396.243,Z 389.64,A -85,B 0,C 180,E1 -11241.843,E2 -11241.843} C_VEL
LIN {X 0,Y 395.993,Z 395.162,A -85,B 0,C 180,E1 -11243.657,E2 -11243.657} C_VEL
LIN {X 0,Y 395.921,Z 398.048,A -85,B 0,C 180,E1 -11244.908,E2 -11244.908} C_VEL
LIN {X 0,Y 395.802,Z 399.924,A -85,B 0,C 180,E1 -11245.927,E2 -11245.927} C_VEL
LIN {X 0,Y 395.812,Z 401.338,A -85,B 0,C 180,E1 -11246.947,E2 -11246.947} C_VEL
LIN {X 0,Y 395.854,Z 402.348,A -85,B 0,C 180,E1 -11247.965,E2 -11247.965} C_VEL
LIN {X 0,Y 395.813,Z 402.961,A -85,B 0,C 180,E1 -11248.983,E2 -11248.983} C_VEL
LIN {X 0,Y 395.815,Z 403.18,A -85,B 0,C 180,E1 -11250,E2 -11250} C_VEL
LIN {X 0,Y 395.813,Z 402.961,A -85,B 0,C 180,E1 -11251.018,E2 -11251.018} C_VEL
LIN {X 0,Y 395.854,Z 402.349,A -85,B 0,C 180,E1 -11252.035,E2 -11252.035} C_VEL
LIN {X 0,Y 395.812,Z 401.34,A -85,B 0,C 180,E1 -11253.054,E2 -11253.054} C_VEL
LIN {X 0,Y 395.802,Z 399.927,A -85,B 0,C 180,E1 -11254.073,E2 -11254.073} C_VEL
LIN {X 0,Y 395.907,Z 396.963,A -85,B 0,C 180,E1 -11255.603,E2 -11255.603} C_VEL
LIN {X 0,Y 396.062,Z 392.953,A -85,B 0,C 180,E1 -11257.136,E2 -11257.136} C_VEL
LIN {X 0,Y 396.458,Z 386.796,A -85,B 0,C 180,E1 -11258.923,E2 -11258.923} C_VEL
LIN {X 0,Y 396.917,Z 380.072,A -85,B 0,C 180,E1 -11260.457,E2 -11260.457} C_VEL
LIN {X 0,Y 397.612,Z 371.742,A -85,B 0,C 180,E1 -11261.987,E2 -11261.987} C_VEL
LIN {X 0,Y 398.285,Z 363.208,A -85,B 0,C 180,E1 -11263.262,E2 -11263.262} C_VEL
LIN {X 0,Y 399.133,Z 352.914,A -85,B 0,C 180,E1 -11264.506,E2 -11264.506} C_VEL
LIN {X 0,Y 399.939,Z 342.262,A -85,B 0,C 180,E1 -11265.545,E2 -11265.545} C_VEL
LIN {X 0,Y 400.825,Z 331.062,A -85,B 0,C 180,E1 -11266.409,E2 -11266.409} C_VEL
LIN {X 0,Y 401.098,Z 325.84,A -85,B 0,C 180,E1 -11266.746,E2 -11266.746} C_VEL
LIN {X 0,Y 399.449,Z 313.142,A -85,B 0,C 180,E1 -11267.495,E2 -11267.495} C_VEL
LIN {X 0,Y 397.424,Z 299.94,A -85,B 0,C 180,E1 -11268.069,E2 -11268.069} C_VEL
LIN {X 0,Y 396.61,Z 295.158,A -85,B 0,C 180,E1 -11268.232,E2 -11268.232} C_VEL
LIN {X 0,Y 397.074,Z 286.691,A -85,B 0,C 180,E1 -11271.82,E2 -11271.82} C_VEL
LIN {X 0,Y 397.524,Z 278.905,A -85,B 0,C 180,E1 -11275.107,E2 -11275.107} C_VEL
LIN {X 0,Y 398.127,Z 271.006,A -85,B 0,C 180,E1 -11278.465,E2 -11278.465} C_VEL
LIN {X 0,Y 398.835,Z 262.334,A -85,B 0,C 180,E1 -11282.239,E2 -11282.239} C_VEL
LIN {X 0,Y 399.432,Z 255.211,A -85,B 0,C 180,E1 -11285.496,E2 -11285.496} C_VEL
LIN {X 0,Y 399.44,Z 252.618,A -85,B 0,C 180,E1 -11286.743,E2 -11286.743} C_VEL
LIN {X 0,Y 398.64,Z 247.416,A -85,B 0,C 180,E1 -11289.397,E2 -11289.397} C_VEL
LIN {X 0,Y 397.502,Z 241.078,A -85,B 0,C 180,E1 -11292.848,E2 -11292.848} C_VEL
LIN {X 0,Y 397.121,Z 239.026,A -85,B 0,C 180,E1 -11294.086,E2 -11294.086} C_VEL
LIN {X 0,Y 397.101,Z 239.021,A -85,B 0,C 180,E1 -11296.522,E2 -11296.522} C_VEL
LIN {X 0,Y 397.089,Z 239.022,A -85,B 0,C 180,E1 -11300.42,E2 -11300.42} C_VEL
LIN {X 0,Y 397.1,Z 239.02,A -85,B 0,C 180,E1 -11303.005,E2 -11303.005} C_VEL
LIN {X 0,Y 397.122,Z 239.02,A -85,B 0,C 180,E1 -11306.282,E2 -11306.282} C_VEL
LIN {X 0,Y 397.103,Z 239.022,A -85,B 0,C 180,E1 -11310.137,E2 -11310.137} C_VEL
LIN {X 0,Y 397.085,Z 239.021,A -85,B 0,C 180,E1 -11313.738,E2 -11313.738} C_VEL
LIN {X 0,Y 397.103,Z 239.017,A -85,B 0,C 180,E1 -11317.085,E2 -11317.085} C_VEL
LIN {X 0,Y 397.152,Z 239.015,A -85,B 0,C 180,E1 -11320.353,E2 -11320.353} C_VEL
LIN {X 0,Y 397.17,Z 239.012,A -85,B 0,C 180,E1 -11323.553,E2 -11323.553} C_VEL
LIN {X 0,Y 397.233,Z 239.001,A -85,B 0,C 180,E1 -11326.703,E2 -11326.703} C_VEL
LIN {X 0,Y 397.21,Z 239.01,A -85,B 0,C 180,E1 -11329.809,E2 -11329.809} C_VEL
LIN {X 0,Y 397.338,Z 238.989,A -85,B 0,C 180,E1 -11332.888,E2 -11332.888} C_VEL
LIN {X 0,Y 397.256,Z 238.999,A -85,B 0,C 180,E1 -11334.925,E2 -11334.925} C_VEL
LIN {X 0,Y 397.453,Z 238.976,A -85,B 0,C 180,E1 -11337.973,E2 -11337.973} C_VEL
LIN {X 0,Y 397.447,Z 238.975,A -85,B 0,C 180,E1 -11342.027,E2 -11342.027} C_VEL
LIN {X 0,Y 397.336,Z 238.989,A -85,B 0,C 180,E1 -11346.643,E2 -11346.643} C_VEL
LIN {X 0,Y 397.24,Z 239.005,A -85,B 0,C 180,E1 -11349.162,E2 -11349.162} C_VEL
LIN {X 0,Y 397.224,Z 239.003,A -85,B 0,C 180,E1 -11352.258,E2 -11352.258} C_VEL
LIN {X 0,Y 397.177,Z 239.01,A -85,B 0,C 180,E1 -11355.392,E2 -11355.392} C_VEL
LIN {X 0,Y 397.161,Z 239.013,A -85,B 0,C 180,E1 -11358.574,E2 -11358.574} C_VEL
LIN {X 0,Y 397.1,Z 239.018,A -85,B 0,C 180,E1 -11361.818,E2 -11361.818} C_VEL
LIN {X 0,Y 397.127,Z 239.017,A -85,B 0,C 180,E1 -11365.134,E2 -11365.134} C_VEL
LIN {X 0,Y 397.075,Z 239.026,A -85,B 0,C 180,E1 -11368.547,E2 -11368.547} C_VEL
LIN {X 0,Y 397.084,Z 239.02,A -85,B 0,C 180,E1 -11371.836,E2 -11371.836} C_VEL
LIN {X 0,Y 397.129,Z 239.019,A -85,B 0,C 180,E1 -11374.493,E2 -11374.493} C_VEL
LIN {X 0,Y 397.102,Z 239.023,A -85,B 0,C 180,E1 -11378.275,E2 -11378.275} C_VEL
LIN {X 0,Y 397.09,Z 239.02,A -85,B 0,C 180,E1 -11380.909,E2 -11380.909} C_VEL
LIN {X 0,Y 397.103,Z 239.019,A -85,B 0,C 180,E1 -11383.648,E2 -11383.648} C_VEL
LIN {X 0,Y 397.104,Z 239.019,A -85,B 0,C 180,E1 -11386.521,E2 -11386.521} C_VEL
LIN {X 0,Y 397.115,Z 239.018,A -85,B 0,C 180,E1 -11390.422,E2 -11390.422} C_VEL
LIN {X 0,Y 397.086,Z 239.02,A -85,B 0,C 180,E1 -11393.003,E2 -11393.003} C_VEL
LIN {X 0,Y 396.916,Z 239.045,A -85,B 0,C 180,E1 -11395.485,E2 -11395.485} C_VEL
LIN {X 0,Y 396.592,Z 239.087,A -85,B 0,C 180,E1 -11398.278,E2 -11398.278} C_VEL
LIN {X 0,Y 396.5,Z 241.93,A -85,B 0,C 180,E1 -11401.407,E2 -11401.407} C_VEL
LIN {X 0,Y 396.411,Z 245.129,A -85,B 0,C 180,E1 -11404.817,E2 -11404.817} C_VEL
LIN {X 0,Y 396.292,Z 248.428,A -85,B 0,C 180,E1 -11408.135,E2 -11408.135} C_VEL
LIN {X 0,Y 396.267,Z 251.902,A -85,B 0,C 180,E1 -11411.383,E2 -11411.383} C_VEL
LIN {X 0,Y 396.28,Z 252.426,A -85,B 0,C 180,E1 -11411.858,E2 -11411.858} C_VEL
LIN {X 0,Y 400.141,Z 266.677,A -85,B 0,C 180,E1 -11412.561,E2 -11412.561} C_VEL
LIN {X 0,Y 402.054,Z 276.321,A -85,B 0,C 180,E1 -11413.152,E2 -11413.152} C_VEL
LIN {X 0,Y 401.437,Z 287.368,A -85,B 0,C 180,E1 -11413.863,E2 -11413.863} C_VEL
LIN {X 0,Y 400.745,Z 298.098,A -85,B 0,C 180,E1 -11414.748,E2 -11414.748} C_VEL
LIN {X 0,Y 400.034,Z 307.957,A -85,B 0,C 180,E1 -11415.761,E2 -11415.761} C_VEL
LIN {X 0,Y 399.169,Z 317.899,A -85,B 0,C 180,E1 -11417.027,E2 -11417.027} C_VEL
LIN {X 0,Y 398.364,Z 327.498,A -85,B 0,C 180,E1 -11418.552,E2 -11418.552} C_VEL
LIN {X 0,Y 397.62,Z 335.157,A -85,B 0,C 180,E1 -11420.076,E2 -11420.076} C_VEL
LIN {X 0,Y 396.976,Z 342.176,A -85,B 0,C 180,E1 -11421.858,E2 -11421.858} C_VEL
LIN {X 0,Y 396.646,Z 346.845,A -85,B 0,C 180,E1 -11423.386,E2 -11423.386} C_VEL
LIN {X 0,Y 396.274,Z 350.426,A -85,B 0,C 180,E1 -11424.912,E2 -11424.912} C_VEL
LIN {X 0,Y 396.284,Z 352.264,A -85,B 0,C 180,E1 -11425.932,E2 -11425.932} C_VEL
LIN {X 0,Y 396.155,Z 353.657,A -85,B 0,C 180,E1 -11426.949,E2 -11426.949} C_VEL
LIN {X 0,Y 395.922,Z 355.262,A -85,B 0,C 180,E1 -11428.983,E2 -11428.983} C_VEL
LIN {X 0,Y 395.912,Z 355.493,A -85,B 0,C 180,E1 -11430,E2 -11430} C_VEL
LIN {X 0,Y 395.999,Z 354.724,A -85,B 0,C 180,E1 -11432.034,E2 -11432.034} C_VEL
LIN {X 0,Y 396.148,Z 353.76,A -85,B 0,C 180,E1 -11433.051,E2 -11433.051} C_VEL
LIN {X 0,Y 396.279,Z 352.412,A -85,B 0,C 180,E1 -11434.068,E2 -11434.068} C_VEL
LIN {X 0,Y 396.318,Z 349.577,A -85,B 0,C 180,E1 -11435.597,E2 -11435.597} C_VEL
LIN {X 0,Y 396.721,Z 345.425,A -85,B 0,C 180,E1 -11437.227,E2 -11437.227} C_VEL
LIN {X 0,Y 397.086,Z 340.732,A -85,B 0,C 180,E1 -11438.652,E2 -11438.652} C_VEL
LIN {X 0,Y 397.718,Z 334.45,A -85,B 0,C 180,E1 -11440.178,E2 -11440.178} C_VEL
LIN {X 0,Y 398.404,Z 326.588,A -85,B 0,C 180,E1 -11441.704,E2 -11441.704} C_VEL
LIN {X 0,Y 399.133,Z 318.566,A -85,B 0,C 180,E1 -11442.974,E2 -11442.974} C_VEL
LIN {X 0,Y 400.016,Z 308.767,A -85,B 0,C 180,E1 -11444.239,E2 -11444.239} C_VEL
LIN {X 0,Y 400.744,Z 298.64,A -85,B 0,C 180,E1 -11445.299,E2 -11445.299} C_VEL
LIN {X 0,Y 401.034,Z 294.563,A -85,B 0,C 180,E1 -11445.662,E2 -11445.662} C_VEL
LIN {X 0,Y 400.767,Z 289.528,A -85,B 0,C 180,E1 -11446.111,E2 -11446.111} C_VEL
LIN {X 0,Y 399.533,Z 284.559,A -85,B 0,C 180,E1 -11446.55,E2 -11446.55} C_VEL
LIN {X 0,Y 395.681,Z 274.606,A -85,B 0,C 180,E1 -11447.364,E2 -11447.364} C_VEL
LIN {X 0,Y 393.259,Z 267.609,A -85,B 0,C 180,E1 -11447.832,E2 -11447.832} C_VEL
LIN {X 0,Y 389.756,Z 254.884,A -85,B 0,C 180,E1 -11448.49,E2 -11448.49} C_VEL
LIN {X 0,Y 389.219,Z 252.777,A -85,B 0,C 180,E1 -11448.591,E2 -11448.591} C_VEL
LIN {X 0,Y 389.233,Z 250.054,A -85,B 0,C 180,E1 -11451.169,E2 -11451.169} C_VEL
LIN {X 0,Y 389.32,Z 246.7,A -85,B 0,C 180,E1 -11454.532,E2 -11454.532} C_VEL
LIN {X 0,Y 389.401,Z 243.446,A -85,B 0,C 180,E1 -11457.986,E2 -11457.986} C_VEL
LIN {X 0,Y 389.514,Z 241.271,A -85,B 0,C 180,E1 -11460.345,E2 -11460.345} C_VEL
LIN {X 0,Y 389.564,Z 239.963,A -85,B 0,C 180,E1 -11462.014,E2 -11462.014} C_VEL
LIN {X 0,Y 389.924,Z 239.912,A -85,B 0,C 180,E1 -11465.224,E2 -11465.224} C_VEL
LIN {X 0,Y 390.037,Z 239.9,A -85,B 0,C 180,E1 -11467.781,E2 -11467.781} C_VEL
LIN {X 0,Y 390.057,Z 239.896,A -85,B 0,C 180,E1 -11470.821,E2 -11470.821} C_VEL
LIN {X 0,Y 390.056,Z 239.9,A -85,B 0,C 180,E1 -11473.886,E2 -11473.886} C_VEL
LIN {X 0,Y 390.057,Z 239.895,A -85,B 0,C 180,E1 -11476.789,E2 -11476.789} C_VEL
LIN {X 0,Y 390.058,Z 239.898,A -85,B 0,C 180,E1 -11479.56,E2 -11479.56} C_VEL
LIN {X 0,Y 390.044,Z 239.897,A -85,B 0,C 180,E1 -11482.45,E2 -11482.45} C_VEL
LIN {X 0,Y 390.07,Z 239.896,A -85,B 0,C 180,E1 -11485.975,E2 -11485.975} C_VEL
LIN {X 0,Y 390.039,Z 239.902,A -85,B 0,C 180,E1 -11489.7,E2 -11489.7} C_VEL
LIN {X 0,Y 390.051,Z 239.9,A -85,B 0,C 180,E1 -11493.227,E2 -11493.227} C_VEL
LIN {X 0,Y 390.069,Z 239.895,A -85,B 0,C 180,E1 -11496.764,E2 -11496.764} C_VEL
LIN {X 0,Y 390.106,Z 239.889,A -85,B 0,C 180,E1 -11499.983,E2 -11499.983} C_VEL
LIN {X 0,Y 390.139,Z 239.889,A -85,B 0,C 180,E1 -11503.248,E2 -11503.248} C_VEL
LIN {X 0,Y 390.197,Z 239.88,A -85,B 0,C 180,E1 -11506.562,E2 -11506.562} C_VEL
LIN {X 0,Y 390.208,Z 239.881,A -85,B 0,C 180,E1 -11510.671,E2 -11510.671} C_VEL
LIN {X 0,Y 390.32,Z 239.867,A -85,B 0,C 180,E1 -11512.759,E2 -11512.759} C_VEL
LIN {X 0,Y 390.222,Z 239.88,A -85,B 0,C 180,E1 -11514.833,E2 -11514.833} C_VEL
LIN {X 0,Y 390.413,Z 239.851,A -85,B 0,C 180,E1 -11517.937,E2 -11517.937} C_VEL
LIN {X 0,Y 390.42,Z 239.852,A -85,B 0,C 180,E1 -11522.063,E2 -11522.063} C_VEL
LIN {X 0,Y 390.32,Z 239.867,A -85,B 0,C 180,E1 -11526.202,E2 -11526.202} C_VEL
LIN {X 0,Y 390.192,Z 239.878,A -85,B 0,C 180,E1 -11529.329,E2 -11529.329} C_VEL
LIN {X 0,Y 390.197,Z 239.878,A -85,B 0,C 180,E1 -11533.438,E2 -11533.438} C_VEL
LIN {X 0,Y 390.151,Z 239.884,A -85,B 0,C 180,E1 -11537.308,E2 -11537.308} C_VEL
LIN {X 0,Y 390.09,Z 239.892,A -85,B 0,C 180,E1 -11540.47,E2 -11540.47} C_VEL
LIN {X 0,Y 390.064,Z 239.896,A -85,B 0,C 180,E1 -11543.353,E2 -11543.353} C_VEL
LIN {X 0,Y 390.044,Z 239.896,A -85,B 0,C 180,E1 -11546.773,E2 -11546.773} C_VEL
LIN {X 0,Y 390.038,Z 239.898,A -85,B 0,C 180,E1 -11550.3,E2 -11550.3} C_VEL
LIN {X 0,Y 390.07,Z 239.895,A -85,B 0,C 180,E1 -11554.025,E2 -11554.025} C_VEL
LIN {X 0,Y 390.041,Z 239.902,A -85,B 0,C 180,E1 -11557.55,E2 -11557.55} C_VEL
LIN {X 0,Y 390.018,Z 239.902,A -85,B 0,C 180,E1 -11560.815,E2 -11560.815} C_VEL
LIN {X 0,Y 390.053,Z 239.899,A -85,B 0,C 180,E1 -11563.886,E2 -11563.886} C_VEL
LIN {X 0,Y 390.065,Z 239.951,A -85,B 0,C 180,E1 -11565.583,E2 -11565.583} C_VEL
LIN {X 0,Y 391.18,Z 245.851,A -85,B 0,C 180,E1 -11568.989,E2 -11568.989} C_VEL
LIN {X 0,Y 392.184,Z 251.576,A -85,B 0,C 180,E1 -11572.045,E2 -11572.045} C_VEL
LIN {X 0,Y 392.465,Z 255.026,A -85,B 0,C 180,E1 -11573.776,E2 -11573.776} C_VEL
LIN {X 0,Y 392.087,Z 260.254,A -85,B 0,C 180,E1 -11576.244,E2 -11576.244} C_VEL
LIN {X 0,Y 391.63,Z 265.499,A -85,B 0,C 180,E1 -11578.64,E2 -11578.64} C_VEL
LIN {X 0,Y 390.973,Z 273.36,A -85,B 0,C 180,E1 -11582.136,E2 -11582.136} C_VEL
LIN {X 0,Y 390.375,Z 281.178,A -85,B 0,C 180,E1 -11585.539,E2 -11585.539} C_VEL
LIN {X 0,Y 389.905,Z 288.883,A -85,B 0,C 180,E1 -11588.869,E2 -11588.869} C_VEL
LIN {X 0,Y 389.566,Z 294.798,A -85,B 0,C 180,E1 -11591.426,E2 -11591.426} C_VEL
LIN {X 0,Y 391.844,Z 308.324,A -85,B 0,C 180,E1 -11591.961,E2 -11591.961} C_VEL
LIN {X 0,Y 393.442,Z 320.584,A -85,B 0,C 180,E1 -11592.629,E2 -11592.629} C_VEL
LIN {X 0,Y 394.149,Z 327.497,A -85,B 0,C 180,E1 -11593.087,E2 -11593.087} C_VEL
LIN {X 0,Y 393.324,Z 338.876,A -85,B 0,C 180,E1 -11593.921,E2 -11593.921} C_VEL
LIN {X 0,Y 392.398,Z 349.896,A -85,B 0,C 180,E1 -11594.948,E2 -11594.948} C_VEL
LIN {X 0,Y 391.591,Z 359.763,A -85,B 0,C 180,E1 -11596.099,E2 -11596.099} C_VEL
LIN {X 0,Y 390.796,Z 369.729,A -85,B 0,C 180,E1 -11597.537,E2 -11597.537} C_VEL
LIN {X 0,Y 389.968,Z 378.403,A -85,B 0,C 180,E1 -11599.092,E2 -11599.092} C_VEL
LIN {X 0,Y 389.453,Z 385.35,A -85,B 0,C 180,E1 -11600.653,E2 -11600.653} C_VEL
LIN {X 0,Y 389.076,Z 390.922,A -85,B 0,C 180,E1 -11602.214,E2 -11602.214} C_VEL
LIN {X 0,Y 388.833,Z 396.077,A -85,B 0,C 180,E1 -11604.096,E2 -11604.096} C_VEL
LIN {X 0,Y 388.729,Z 399.498,A -85,B 0,C 180,E1 -11605.853,E2 -11605.853} C_VEL
LIN {X 0,Y 388.788,Z 401.922,A -85,B 0,C 180,E1 -11607.928,E2 -11607.928} C_VEL
LIN {X 0,Y 388.743,Z 402.535,A -85,B 0,C 180,E1 -11608.964,E2 -11608.964} C_VEL
LIN {X 0,Y 388.742,Z 402.754,A -85,B 0,C 180,E1 -11610,E2 -11610} C_VEL
LIN {X 0,Y 388.743,Z 402.535,A -85,B 0,C 180,E1 -11611.036,E2 -11611.036} C_VEL
LIN {X 0,Y 388.788,Z 401.923,A -85,B 0,C 180,E1 -11612.072,E2 -11612.072} C_VEL
LIN {X 0,Y 388.729,Z 399.499,A -85,B 0,C 180,E1 -11614.147,E2 -11614.147} C_VEL
LIN {X 0,Y 388.831,Z 396.082,A -85,B 0,C 180,E1 -11615.901,E2 -11615.901} C_VEL
LIN {X 0,Y 389.078,Z 390.916,A -85,B 0,C 180,E1 -11617.786,E2 -11617.786} C_VEL
LIN {X 0,Y 389.453,Z 385.344,A -85,B 0,C 180,E1 -11619.347,E2 -11619.347} C_VEL
LIN {X 0,Y 389.968,Z 378.394,A -85,B 0,C 180,E1 -11620.908,E2 -11620.908} C_VEL
LIN {X 0,Y 390.795,Z 369.716,A -85,B 0,C 180,E1 -11622.463,E2 -11622.463} C_VEL
LIN {X 0,Y 391.536,Z 361.069,A -85,B 0,C 180,E1 -11623.725,E2 -11623.725} C_VEL
LIN {X 0,Y 392.288,Z 351.058,A -85,B 0,C 180,E1 -11624.924,E2 -11624.924} C_VEL
LIN {X 0,Y 393.176,Z 340.394,A -85,B 0,C 180,E1 -11625.952,E2 -11625.952} C_VEL
LIN {X 0,Y 394.092,Z 329.145,A -85,B 0,C 180,E1 -11626.803,E2 -11626.803} C_VEL
LIN {X 0,Y 393.932,Z 324.021,A -85,B 0,C 180,E1 -11627.145,E2 -11627.145} C_VEL
LIN {X 0,Y 392.351,Z 311.774,A -85,B 0,C 180,E1 -11627.862,E2 -11627.862} C_VEL
LIN {X 0,Y 390.129,Z 298.252,A -85,B 0,C 180,E1 -11628.455,E2 -11628.455} C_VEL
LIN {X 0,Y 389.568,Z 294.737,A -85,B 0,C 180,E1 -11628.574,E2 -11628.574} C_VEL
LIN {X 0,Y 390.049,Z 286.313,A -85,B 0,C 180,E1 -11632.234,E2 -11632.234} C_VEL
LIN {X 0,Y 390.619,Z 277.867,A -85,B 0,C 180,E1 -11635.894,E2 -11635.894} C_VEL
LIN {X 0,Y 391.169,Z 270.69,A -85,B 0,C 180,E1 -11639.019,E2 -11639.019} C_VEL
LIN {X 0,Y 391.872,Z 262.764,A -85,B 0,C 180,E1 -11642.55,E2 -11642.55} C_VEL
LIN {X 0,Y 392.449,Z 256.272,A -85,B 0,C 180,E1 -11645.593,E2 -11645.593} C_VEL
LIN {X 0,Y 392.261,Z 252.374,A -85,B 0,C 180,E1 -11647.53,E2 -11647.53} C_VEL
LIN {X 0,Y 391.182,Z 245.854,A -85,B 0,C 180,E1 -11651.012,E2 -11651.012} C_VEL
LIN {X 0,Y 390.094,Z 239.899,A -85,B 0,C 180,E1 -11654.432,E2 -11654.432} C_VEL
LIN {X 0,Y 390.035,Z 239.903,A -85,B 0,C 180,E1 -11657.628,E2 -11657.628} C_VEL
LIN {X 0,Y 390.061,Z 239.898,A -85,B 0,C 180,E1 -11660.904,E2 -11660.904} C_VEL
LIN {X 0,Y 390.088,Z 239.895,A -85,B 0,C 180,E1 -11664.793,E2 -11664.793} C_VEL
LIN {X 0,Y 390.027,Z 239.904,A -85,B 0,C 180,E1 -11668.496,E2 -11668.496} C_VEL
LIN {X 0,Y 390.028,Z 239.902,A -85,B 0,C 180,E1 -11672.063,E2 -11672.063} C_VEL
LIN {X 0,Y 390.046,Z 239.897,A -85,B 0,C 180,E1 -11675.517,E2 -11675.517} C_VEL
LIN {X 0,Y 390.059,Z 239.895,A -85,B 0,C 180,E1 -11678.878,E2 -11678.878} C_VEL
LIN {X 0,Y 390.132,Z 239.891,A -85,B 0,C 180,E1 -11682.167,E2 -11682.167} C_VEL
LIN {X 0,Y 390.147,Z 239.885,A -85,B 0,C 180,E1 -11685.393,E2 -11685.393} C_VEL
LIN {X 0,Y 390.141,Z 239.884,A -85,B 0,C 180,E1 -11688.571,E2 -11688.571} C_VEL
LIN {X 0,Y 390.274,Z 239.871,A -85,B 0,C 180,E1 -11692.072,E2 -11692.072} C_VEL
LIN {X 0,Y 390.227,Z 239.874,A -85,B 0,C 180,E1 -11694.834,E2 -11694.834} C_VEL
LIN {X 0,Y 390.422,Z 239.852,A -85,B 0,C 180,E1 -11697.937,E2 -11697.937} C_VEL
LIN {X 0,Y 390.415,Z 239.851,A -85,B 0,C 180,E1 -11702.063,E2 -11702.063} C_VEL
LIN {X 0,Y 390.29,Z 239.866,A -85,B 0,C 180,E1 -11706.637,E2 -11706.637} C_VEL
LIN {X 0,Y 390.198,Z 239.883,A -85,B 0,C 180,E1 -11709.329,E2 -11709.329} C_VEL
LIN {X 0,Y 390.175,Z 239.881,A -85,B 0,C 180,E1 -11712.483,E2 -11712.483} C_VEL
LIN {X 0,Y 390.139,Z 239.885,A -85,B 0,C 180,E1 -11715.677,E2 -11715.677} C_VEL
LIN {X 0,Y 390.106,Z 239.894,A -85,B 0,C 180,E1 -11718.922,E2 -11718.922} C_VEL
LIN {X 0,Y 390.042,Z 239.898,A -85,B 0,C 180,E1 -11722.234,E2 -11722.234} C_VEL
LIN {X 0,Y 390.071,Z 239.893,A -85,B 0,C 180,E1 -11725.727,E2 -11725.727} C_VEL
LIN {X 0,Y 390.032,Z 239.899,A -85,B 0,C 180,E1 -11729.112,E2 -11729.112} C_VEL
LIN {X 0,Y 390.046,Z 239.9,A -85,B 0,C 180,E1 -11732.721,E2 -11732.721} C_VEL
LIN {X 0,Y 390.059,Z 239.896,A -85,B 0,C 180,E1 -11735.825,E2 -11735.825} C_VEL
LIN {X 0,Y 390.07,Z 239.894,A -85,B 0,C 180,E1 -11739.217,E2 -11739.217} C_VEL
LIN {X 0,Y 390.043,Z 239.901,A -85,B 0,C 180,E1 -11742.373,E2 -11742.373} C_VEL
LIN {X 0,Y 390.047,Z 239.896,A -85,B 0,C 180,E1 -11745.354,E2 -11745.354} C_VEL
LIN {X 0,Y 390.028,Z 239.903,A -85,B 0,C 180,E1 -11748.186,E2 -11748.186} C_VEL
LIN {X 0,Y 390.089,Z 239.891,A -85,B 0,C 180,E1 -11750.907,E2 -11750.907} C_VEL
LIN {X 0,Y 389.971,Z 239.908,A -85,B 0,C 180,E1 -11754.193,E2 -11754.193} C_VEL
LIN {X 0,Y 389.635,Z 239.953,A -85,B 0,C 180,E1 -11757.24,E2 -11757.24} C_VEL
LIN {X 0,Y 389.526,Z 240.102,A -85,B 0,C 180,E1 -11758.45,E2 -11758.45} C_VEL
LIN {X 0,Y 389.434,Z 243.339,A -85,B 0,C 180,E1 -11762.016,E2 -11762.016} C_VEL
LIN {X 0,Y 389.321,Z 246.588,A -85,B 0,C 180,E1 -11765.468,E2 -11765.468} C_VEL
LIN {X 0,Y 389.235,Z 249.95,A -85,B 0,C 180,E1 -11768.831,E2 -11768.831} C_VEL
LIN {X 0,Y 389.232,Z 252.834,A -85,B 0,C 180,E1 -11771.511,E2 -11771.511} C_VEL
LIN {X 0,Y 393.155,Z 267.338,A -85,B 0,C 180,E1 -11772.251,E2 -11772.251} C_VEL
LIN {X 0,Y 395.265,Z 277.403,A -85,B 0,C 180,E1 -11772.892,E2 -11772.892} C_VEL
LIN {X 0,Y 394.569,Z 289.539,A -85,B 0,C 180,E1 -11773.708,E2 -11773.708} C_VEL
LIN {X 0,Y 393.771,Z 301.248,A -85,B 0,C 180,E1 -11774.746,E2 -11774.746} C_VEL
LIN {X 0,Y 392.957,Z 311.578,A -85,B 0,C 180,E1 -11775.896,E2 -11775.896} C_VEL
LIN {X 0,Y 392.131,Z 320.094,A -85,B 0,C 180,E1 -11777.054,E2 -11777.054} C_VEL
LIN {X 0,Y 391.428,Z 327.927,A -85,B 0,C 180,E1 -11778.346,E2 -11778.346} C_VEL
LIN {X 0,Y 390.648,Z 335.585,A -85,B 0,C 180,E1 -11779.897,E2 -11779.897} C_VEL
LIN {X 0,Y 389.97,Z 342.604,A -85,B 0,C 180,E1 -11781.71,E2 -11781.71} C_VEL
LIN {X 0,Y 389.63,Z 346.813,A -85,B 0,C 180,E1 -11783.096,E2 -11783.096} C_VEL
LIN {X 0,Y 389.208,Z 350.854,A -85,B 0,C 180,E1 -11784.82,E2 -11784.82} C_VEL
LIN {X 0,Y 389.214,Z 352.692,A -85,B 0,C 180,E1 -11785.858,E2 -11785.858} C_VEL
LIN {X 0,Y 389.098,Z 354.083,A -85,B 0,C 180,E1 -11786.894,E2 -11786.894} C_VEL
LIN {X 0,Y 388.848,Z 355.688,A -85,B 0,C 180,E1 -11788.964,E2 -11788.964} C_VEL
LIN {X 0,Y 388.835,Z 355.92,A -85,B 0,C 180,E1 -11790,E2 -11790} C_VEL
LIN {X 0,Y 388.933,Z 355.149,A -85,B 0,C 180,E1 -11792.071,E2 -11792.071} C_VEL
LIN {X 0,Y 389.091,Z 354.185,A -85,B 0,C 180,E1 -11793.106,E2 -11793.106} C_VEL
LIN {X 0,Y 389.208,Z 352.838,A -85,B 0,C 180,E1 -11794.142,E2 -11794.142} C_VEL
LIN {X 0,Y 389.275,Z 350.002,A -85,B 0,C 180,E1 -11795.699,E2 -11795.699} C_VEL
LIN {X 0,Y 389.66,Z 346.138,A -85,B 0,C 180,E1 -11797.253,E2 -11797.253} C_VEL
LIN {X 0,Y 390.091,Z 341.156,A -85,B 0,C 180,E1 -11798.809,E2 -11798.809} C_VEL
LIN {X 0,Y 390.743,Z 334.875,A -85,B 0,C 180,E1 -11800.362,E2 -11800.362} C_VEL
LIN {X 0,Y 391.471,Z 327.012,A -85,B 0,C 180,E1 -11801.915,E2 -11801.915} C_VEL
LIN {X 0,Y 392.238,Z 318.989,A -85,B 0,C 180,E1 -11803.206,E2 -11803.206} C_VEL
LIN {X 0,Y 393.148,Z 309.19,A -85,B 0,C 180,E1 -11804.493,E2 -11804.493} C_VEL
LIN {X 0,Y 394.006,Z 298.164,A -85,B 0,C 180,E1 -11805.652,E2 -11805.652} C_VEL
LIN {X 0,Y 394.728,Z 287.347,A -85,B 0,C 180,E1 -11806.551,E2 -11806.551} C_VEL
LIN {X 0,Y 395.202,Z 276.341,A -85,B 0,C 180,E1 -11807.274,E2 -11807.274} C_VEL
LIN {X 0,Y 393.259,Z 267.609,A -85,B 0,C 180,E1 -11807.832,E2 -11807.832} C_VEL
LIN {X 0,Y 391.759,Z 265.585,A -85,B 0,C 180,E1 -11807.998,E2 -11807.998} C_VEL
LIN {X 0,Y 385.384,Z 262.138,A -85,B 0,C 180,E1 -11808.467,E2 -11808.467} C_VEL
LIN {X 0,Y 384.187,Z 260.309,A -85,B 0,C 180,E1 -11808.598,E2 -11808.598} C_VEL
LIN {X 0,Y 382.163,Z 253.19,A -85,B 0,C 180,E1 -11808.955,E2 -11808.955} C_VEL
LIN {X 0,Y 382.199,Z 250.454,A -85,B 0,C 180,E1 -11811.578,E2 -11811.578} C_VEL
LIN {X 0,Y 382.271,Z 247.074,A -85,B 0,C 180,E1 -11815.015,E2 -11815.015} C_VEL
LIN {X 0,Y 382.369,Z 243.762,A -85,B 0,C 180,E1 -11818.547,E2 -11818.547} C_VEL
LIN {X 0,Y 382.468,Z 241.596,A -85,B 0,C 180,E1 -11820.965,E2 -11820.965} C_VEL
LIN {X 0,Y 382.551,Z 240.836,A -85,B 0,C 180,E1 -11822.319,E2 -11822.319} C_VEL
LIN {X 0,Y 382.806,Z 240.801,A -85,B 0,C 180,E1 -11824.69,E2 -11824.69} C_VEL
LIN {X 0,Y 382.978,Z 240.777,A -85,B 0,C 180,E1 -11827.271,E2 -11827.271} C_VEL
LIN {X 0,Y 383.009,Z 240.777,A -85,B 0,C 180,E1 -11829.958,E2 -11829.958} C_VEL
LIN {X 0,Y 383.007,Z 240.773,A -85,B 0,C 180,E1 -11832.778,E2 -11832.778} C_VEL
LIN {X 0,Y 382.999,Z 240.778,A -85,B 0,C 180,E1 -11835.789,E2 -11835.789} C_VEL
LIN {X 0,Y 382.987,Z 240.775,A -85,B 0,C 180,E1 -11838.796,E2 -11838.796} C_VEL
LIN {X 0,Y 382.999,Z 240.777,A -85,B 0,C 180,E1 -11842.097,E2 -11842.097} C_VEL
LIN {X 0,Y 383.02,Z 240.774,A -85,B 0,C 180,E1 -11845.332,E2 -11845.332} C_VEL
LIN {X 0,Y 383.011,Z 240.776,A -85,B 0,C 180,E1 -11847.85,E2 -11847.85} C_VEL
LIN {X 0,Y 382.983,Z 240.782,A -85,B 0,C 180,E1 -11851.503,E2 -11851.503} C_VEL
LIN {X 0,Y 383.02,Z 240.775,A -85,B 0,C 180,E1 -11855.037,E2 -11855.037} C_VEL
LIN {X 0,Y 382.995,Z 240.775,A -85,B 0,C 180,E1 -11858.469,E2 -11858.469} C_VEL
LIN {X 0,Y 383.055,Z 240.767,A -85,B 0,C 180,E1 -11861.826,E2 -11861.826} C_VEL
LIN {X 0,Y 383.109,Z 240.766,A -85,B 0,C 180,E1 -11865.118,E2 -11865.118} C_VEL
LIN {X 0,Y 383.101,Z 240.763,A -85,B 0,C 180,E1 -11868.358,E2 -11868.358} C_VEL
LIN {X 0,Y 383.306,Z 240.736,A -85,B 0,C 180,E1 -11871.933,E2 -11871.933} C_VEL
LIN {X 0,Y 383.195,Z 240.755,A -85,B 0,C 180,E1 -11874.738,E2 -11874.738} C_VEL
LIN {X 0,Y 383.379,Z 240.727,A -85,B 0,C 180,E1 -11877.899,E2 -11877.899} C_VEL
LIN {X 0,Y 383.388,Z 240.728,A -85,B 0,C 180,E1 -11882.101,E2 -11882.101} C_VEL
LIN {X 0,Y 383.275,Z 240.745,A -85,B 0,C 180,E1 -11886.316,E2 -11886.316} C_VEL
LIN {X 0,Y 383.142,Z 240.756,A -85,B 0,C 180,E1 -11889.502,E2 -11889.502} C_VEL
LIN {X 0,Y 383.127,Z 240.759,A -85,B 0,C 180,E1 -11893.536,E2 -11893.536} C_VEL
LIN {X 0,Y 383.097,Z 240.763,A -85,B 0,C 180,E1 -11897.455,E2 -11897.455} C_VEL
LIN {X 0,Y 383.031,Z 240.771,A -85,B 0,C 180,E1 -11900.647,E2 -11900.647} C_VEL
LIN {X 0,Y 383.011,Z 240.778,A -85,B 0,C 180,E1 -11903.809,E2 -11903.809} C_VEL
LIN {X 0,Y 382.983,Z 240.778,A -85,B 0,C 180,E1 -11907.308,E2 -11907.308} C_VEL
LIN {X 0,Y 382.984,Z 240.777,A -85,B 0,C 180,E1 -11910.919,E2 -11910.919} C_VEL
LIN {X 0,Y 383.019,Z 240.772,A -85,B 0,C 180,E1 -11914.668,E2 -11914.668} C_VEL
LIN {X 0,Y 382.995,Z 240.776,A -85,B 0,C 180,E1 -11917.902,E2 -11917.902} C_VEL
LIN {X 0,Y 382.962,Z 240.784,A -85,B 0,C 180,E1 -11921.35,E2 -11921.35} C_VEL
LIN {X 0,Y 382.996,Z 240.78,A -85,B 0,C 180,E1 -11924.303,E2 -11924.303} C_VEL
LIN {X 0,Y 383.048,Z 240.898,A -85,B 0,C 180,E1 -11925.223,E2 -11925.223} C_VEL
LIN {X 0,Y 384.163,Z 246.963,A -85,B 0,C 180,E1 -11928.807,E2 -11928.807} C_VEL
LIN {X 0,Y 385.101,Z 252.266,A -85,B 0,C 180,E1 -11931.697,E2 -11931.697} C_VEL
LIN {X 0,Y 385.479,Z 255.429,A -85,B 0,C 180,E1 -11933.341,E2 -11933.341} C_VEL
LIN {X 0,Y 385.21,Z 259.985,A -85,B 0,C 180,E1 -11935.557,E2 -11935.557} C_VEL
LIN {X 0,Y 384.616,Z 266.516,A -85,B 0,C 180,E1 -11938.616,E2 -11938.616} C_VEL
LIN {X 0,Y 383.923,Z 274.343,A -85,B 0,C 180,E1 -11942.173,E2 -11942.173} C_VEL
LIN {X 0,Y 383.292,Z 282.112,A -85,B 0,C 180,E1 -11945.634,E2 -11945.634} C_VEL
LIN {X 0,Y 382.807,Z 289.758,A -85,B 0,C 180,E1 -11949.023,E2 -11949.023} C_VEL
LIN {X 0,Y 382.513,Z 294.38,A -85,B 0,C 180,E1 -11951.071,E2 -11951.071} C_VEL
LIN {X 0,Y 384.777,Z 307.78,A -85,B 0,C 180,E1 -11951.614,E2 -11951.614} C_VEL
LIN {X 0,Y 386.414,Z 320.44,A -85,B 0,C 180,E1 -11952.321,E2 -11952.321} C_VEL
LIN {X 0,Y 387.278,Z 327.328,A -85,B 0,C 180,E1 -11952.796,E2 -11952.796} C_VEL
LIN {X 0,Y 386.472,Z 338.45,A -85,B 0,C 180,E1 -11953.628,E2 -11953.628} C_VEL
LIN {X 0,Y 385.508,Z 349.469,A -85,B 0,C 180,E1 -11954.672,E2 -11954.672} C_VEL
LIN {X 0,Y 384.63,Z 359.713,A -85,B 0,C 180,E1 -11955.894,E2 -11955.894} C_VEL
LIN {X 0,Y 383.829,Z 369.301,A -85,B 0,C 180,E1 -11957.307,E2 -11957.307} C_VEL
LIN {X 0,Y 382.967,Z 377.975,A -85,B 0,C 180,E1 -11958.89,E2 -11958.89} C_VEL
LIN {X 0,Y 382.428,Z 384.922,A -85,B 0,C 180,E1 -11960.48,E2 -11960.48} C_VEL
LIN {X 0,Y 382.014,Z 390.493,A -85,B 0,C 180,E1 -11962.069,E2 -11962.069} C_VEL
LIN {X 0,Y 381.805,Z 395.015,A -85,B 0,C 180,E1 -11963.719,E2 -11963.719} C_VEL
LIN {X 0,Y 381.752,Z 397.193,A -85,B 0,C 180,E1 -11964.719,E2 -11964.719} C_VEL
LIN {X 0,Y 381.658,Z 399.071,A -85,B 0,C 180,E1 -11965.776,E2 -11965.776} C_VEL
LIN {X 0,Y 381.704,Z 401.496,A -85,B 0,C 180,E1 -11967.89,E2 -11967.89} C_VEL
LIN {X 0,Y 381.676,Z 402.109,A -85,B 0,C 180,E1 -11968.945,E2 -11968.945} C_VEL
LIN {X 0,Y 381.672,Z 402.328,A -85,B 0,C 180,E1 -11970,E2 -11970} C_VEL
LIN {X 0,Y 381.676,Z 402.109,A -85,B 0,C 180,E1 -11971.055,E2 -11971.055} C_VEL
LIN {X 0,Y 381.704,Z 401.496,A -85,B 0,C 180,E1 -11972.111,E2 -11972.111} C_VEL
LIN {X 0,Y 381.658,Z 399.072,A -85,B 0,C 180,E1 -11974.224,E2 -11974.224} C_VEL
LIN {X 0,Y 381.732,Z 396.018,A -85,B 0,C 180,E1 -11975.852,E2 -11975.852} C_VEL
LIN {X 0,Y 381.928,Z 392.093,A -85,B 0,C 180,E1 -11977.401,E2 -11977.401} C_VEL
LIN {X 0,Y 382.334,Z 385.932,A -85,B 0,C 180,E1 -11979.256,E2 -11979.256} C_VEL
LIN {X 0,Y 382.843,Z 379.207,A -85,B 0,C 180,E1 -11980.846,E2 -11980.846} C_VEL
LIN {X 0,Y 383.656,Z 370.879,A -85,B 0,C 180,E1 -11982.43,E2 -11982.43} C_VEL
LIN {X 0,Y 384.434,Z 362.346,A -85,B 0,C 180,E1 -11983.749,E2 -11983.749} C_VEL
LIN {X 0,Y 385.22,Z 352.989,A -85,B 0,C 180,E1 -11984.934,E2 -11984.934} C_VEL
LIN {X 0,Y 386.094,Z 342.829,A -85,B 0,C 180,E1 -11985.981,E2 -11985.981} C_VEL
LIN {X 0,Y 387.175,Z 330.355,A -85,B 0,C 180,E1 -11986.992,E2 -11986.992} C_VEL
LIN {X 0,Y 387.131,Z 325.67,A -85,B 0,C 180,E1 -11987.32,E2 -11987.32} C_VEL
LIN {X 0,Y 385.699,Z 314.222,A -85,B 0,C 180,E1 -11988.045,E2 -11988.045} C_VEL
LIN {X 0,Y 383.68,Z 300.941,A -85,B 0,C 180,E1 -11988.683,E2 -11988.683} C_VEL
LIN {X 0,Y 382.531,Z 294.314,A -85,B 0,C 180,E1 -11988.929,E2 -11988.929} C_VEL
LIN {X 0,Y 383.063,Z 285.942,A -85,B 0,C 180,E1 -11992.662,E2 -11992.662} C_VEL
LIN {X 0,Y 383.703,Z 276.932,A -85,B 0,C 180,E1 -11996.663,E2 -11996.663} C_VEL
LIN {X 0,Y 384.233,Z 270.373,A -85,B 0,C 180,E1 -11999.595,E2 -11999.595} C_VEL
LIN {X 0,Y 384.911,Z 263.21,A -85,B 0,C 180,E1 -12002.87,E2 -12002.87} C_VEL
LIN {X 0,Y 385.449,Z 257.297,A -85,B 0,C 180,E1 -12005.695,E2 -12005.695} C_VEL
LIN {X 0,Y 385.277,Z 253.461,A -85,B 0,C 180,E1 -12007.644,E2 -12007.644} C_VEL
LIN {X 0,Y 384.173,Z 246.964,A -85,B 0,C 180,E1 -12011.192,E2 -12011.192} C_VEL
LIN {X 0,Y 383.016,Z 240.78,A -85,B 0,C 180,E1 -12014.842,E2 -12014.842} C_VEL
LIN {X 0,Y 383.013,Z 240.778,A -85,B 0,C 180,E1 -12017.24,E2 -12017.24} C_VEL
LIN {X 0,Y 382.988,Z 240.779,A -85,B 0,C 180,E1 -12020.419,E2 -12020.419} C_VEL
LIN {X 0,Y 383.027,Z 240.772,A -85,B 0,C 180,E1 -12024.045,E2 -12024.045} C_VEL
LIN {X 0,Y 382.99,Z 240.775,A -85,B 0,C 180,E1 -12027.578,E2 -12027.578} C_VEL
LIN {X 0,Y 382.981,Z 240.782,A -85,B 0,C 180,E1 -12030.299,E2 -12030.299} C_VEL
LIN {X 0,Y 383.006,Z 240.777,A -85,B 0,C 180,E1 -12034.045,E2 -12034.045} C_VEL
LIN {X 0,Y 382.992,Z 240.775,A -85,B 0,C 180,E1 -12037.334,E2 -12037.334} C_VEL
LIN {X 0,Y 383.064,Z 240.767,A -85,B 0,C 180,E1 -12040.716,E2 -12040.716} C_VEL
LIN {X 0,Y 383.085,Z 240.769,A -85,B 0,C 180,E1 -12044.027,E2 -12044.027} C_VEL
LIN {X 0,Y 383.138,Z 240.758,A -85,B 0,C 180,E1 -12047.284,E2 -12047.284} C_VEL
LIN {X 0,Y 383.142,Z 240.756,A -85,B 0,C 180,E1 -12050.498,E2 -12050.498} C_VEL
LIN {X 0,Y 383.277,Z 240.745,A -85,B 0,C 180,E1 -12053.684,E2 -12053.684} C_VEL
LIN {X 0,Y 383.389,Z 240.728,A -85,B 0,C 180,E1 -12057.899,E2 -12057.899} C_VEL
LIN {X 0,Y 383.381,Z 240.727,A -85,B 0,C 180,E1 -12062.101,E2 -12062.101} C_VEL
LIN {X 0,Y 383.25,Z 240.743,A -85,B 0,C 180,E1 -12066.627,E2 -12066.627} C_VEL
LIN {X 0,Y 383.148,Z 240.759,A -85,B 0,C 180,E1 -12069.502,E2 -12069.502} C_VEL
LIN {X 0,Y 383.13,Z 240.759,A -85,B 0,C 180,E1 -12073.536,E2 -12073.536} C_VEL
LIN {X 0,Y 383.08,Z 240.765,A -85,B 0,C 180,E1 -12077.445,E2 -12077.445} C_VEL
LIN {X 0,Y 383.033,Z 240.774,A -85,B 0,C 180,E1 -12080.647,E2 -12080.647} C_VEL
LIN {X 0,Y 383.021,Z 240.771,A -85,B 0,C 180,E1 -12083.808,E2 -12083.808} C_VEL
LIN {X 0,Y 382.991,Z 240.776,A -85,B 0,C 180,E1 -12087.307,E2 -12087.307} C_VEL
LIN {X 0,Y 382.985,Z 240.778,A -85,B 0,C 180,E1 -12090.919,E2 -12090.919} C_VEL
LIN {X 0,Y 383.021,Z 240.775,A -85,B 0,C 180,E1 -12094.668,E2 -12094.668} C_VEL
LIN {X 0,Y 383.001,Z 240.776,A -85,B 0,C 180,E1 -12097.903,E2 -12097.903} C_VEL
LIN {X 0,Y 382.984,Z 240.776,A -85,B 0,C 180,E1 -12101.348,E2 -12101.348} C_VEL
LIN {X 0,Y 382.999,Z 240.778,A -85,B 0,C 180,E1 -12104.303,E2 -12104.303} C_VEL
LIN {X 0,Y 383.013,Z 240.772,A -85,B 0,C 180,E1 -12107.24,E2 -12107.24} C_VEL
LIN {X 0,Y 383.016,Z 240.774,A -85,B 0,C 180,E1 -12110.414,E2 -12110.414} C_VEL
LIN {X 0,Y 382.941,Z 240.787,A -85,B 0,C 180,E1 -12113.855,E2 -12113.855} C_VEL
LIN {X 0,Y 382.677,Z 240.818,A -85,B 0,C 180,E1 -12116.567,E2 -12116.567} C_VEL
LIN {X 0,Y 382.541,Z 240.837,A -85,B 0,C 180,E1 -12117.806,E2 -12117.806} C_VEL
LIN {X 0,Y 382.451,Z 242.133,A -85,B 0,C 180,E1 -12119.733,E2 -12119.733} C_VEL
LIN {X 0,Y 382.343,Z 244.759,A -85,B 0,C 180,E1 -12122.643,E2 -12122.643} C_VEL
LIN {X 0,Y 382.284,Z 246.962,A -85,B 0,C 180,E1 -12124.986,E2 -12124.986} C_VEL
LIN {X 0,Y 382.201,Z 250.35,A -85,B 0,C 180,E1 -12128.422,E2 -12128.422} C_VEL
LIN {X 0,Y 382.179,Z 253.258,A -85,B 0,C 180,E1 -12131.159,E2 -12131.159} C_VEL
LIN {X 0,Y 386.261,Z 267.995,A -85,B 0,C 180,E1 -12131.932,E2 -12131.932} C_VEL
LIN {X 0,Y 388.469,Z 278.405,A -85,B 0,C 180,E1 -12132.617,E2 -12132.617} C_VEL
LIN {X 0,Y 387.785,Z 289.968,A -85,B 0,C 180,E1 -12133.414,E2 -12133.414} C_VEL
LIN {X 0,Y 386.998,Z 300.571,A -85,B 0,C 180,E1 -12134.355,E2 -12134.355} C_VEL
LIN {X 0,Y 386.145,Z 310.95,A -85,B 0,C 180,E1 -12135.507,E2 -12135.507} C_VEL
LIN {X 0,Y 385.236,Z 320.523,A -85,B 0,C 180,E1 -12136.818,E2 -12136.818} C_VEL
LIN {X 0,Y 384.477,Z 328.358,A -85,B 0,C 180,E1 -12138.133,E2 -12138.133} C_VEL
LIN {X 0,Y 383.687,Z 336.013,A -85,B 0,C 180,E1 -12139.712,E2 -12139.712} C_VEL
LIN {X 0,Y 383.134,Z 341.235,A -85,B 0,C 180,E1 -12141.03,E2 -12141.03} C_VEL
LIN {X 0,Y 382.645,Z 346.438,A -85,B 0,C 180,E1 -12142.666,E2 -12142.666} C_VEL
LIN {X 0,Y 382.252,Z 350.228,A -85,B 0,C 180,E1 -12144.196,E2 -12144.196} C_VEL
LIN {X 0,Y 382.146,Z 353.12,A -85,B 0,C 180,E1 -12145.781,E2 -12145.781} C_VEL
LIN {X 0,Y 382.041,Z 354.509,A -85,B 0,C 180,E1 -12146.836,E2 -12146.836} C_VEL
LIN {X 0,Y 381.776,Z 356.114,A -85,B 0,C 180,E1 -12148.945,E2 -12148.945} C_VEL
LIN {X 0,Y 381.76,Z 356.346,A -85,B 0,C 180,E1 -12150,E2 -12150} C_VEL
LIN {X 0,Y 381.869,Z 355.575,A -85,B 0,C 180,E1 -12152.109,E2 -12152.109} C_VEL
LIN {X 0,Y 382.035,Z 354.61,A -85,B 0,C 180,E1 -12153.164,E2 -12153.164} C_VEL
LIN {X 0,Y 382.14,Z 353.264,A -85,B 0,C 180,E1 -12154.219,E2 -12154.219} C_VEL
LIN {X 0,Y 382.236,Z 350.427,A -85,B 0,C 180,E1 -12155.804,E2 -12155.804} C_VEL
LIN {X 0,Y 382.625,Z 346.564,A -85,B 0,C 180,E1 -12157.387,E2 -12157.387} C_VEL
LIN {X 0,Y 383.088,Z 341.581,A -85,B 0,C 180,E1 -12158.971,E2 -12158.971} C_VEL
LIN {X 0,Y 383.761,Z 335.3,A -85,B 0,C 180,E1 -12160.552,E2 -12160.552} C_VEL
LIN {X 0,Y 384.548,Z 327.435,A -85,B 0,C 180,E1 -12162.132,E2 -12162.132} C_VEL
LIN {X 0,Y 385.358,Z 319.411,A -85,B 0,C 180,E1 -12163.446,E2 -12163.446} C_VEL
LIN {X 0,Y 386.3,Z 309.612,A -85,B 0,C 180,E1 -12164.756,E2 -12164.756} C_VEL
LIN {X 0,Y 387.2,Z 298.585,A -85,B 0,C 180,E1 -12165.934,E2 -12165.934} C_VEL
LIN {X 0,Y 387.963,Z 287.766,A -85,B 0,C 180,E1 -12166.848,E2 -12166.848} C_VEL
LIN {X 0,Y 388.439,Z 277.72,A -85,B 0,C 180,E1 -12167.526,E2 -12167.526} C_VEL
LIN {X 0,Y 385.564,Z 265.283,A -85,B 0,C 180,E1 -12168.327,E2 -12168.327} C_VEL
LIN {X 0,Y 384.187,Z 260.309,A -85,B 0,C 180,E1 -12168.598,E2 -12168.598} C_VEL
LIN {X 0,Y 383.045,Z 257.234,A -85,B 0,C 180,E1 -12168.87,E2 -12168.87} C_VEL
LIN {X 0,Y 381.623,Z 254.934,A -85,B 0,C 180,E1 -12169.27,E2 -12169.27} C_VEL
LIN {X 0,Y 379.368,Z 252.682,A -85,B 0,C 180,E1 -12170.015,E2 -12170.015} C_VEL
LIN {X 0,Y 377.29,Z 251.744,A -85,B 0,C 180,E1 -12170.89,E2 -12170.89} C_VEL
LIN {X 0,Y 375.423,Z 250.711,A -85,B 0,C 180,E1 -12172.153,E2 -12172.153} C_VEL
LIN {X 0,Y 375.175,Z 250.08,A -85,B 0,C 180,E1 -12172.798,E2 -12172.798} C_VEL
LIN {X 0,Y 375.245,Z 247.026,A -85,B 0,C 180,E1 -12175.973,E2 -12175.973} C_VEL
LIN {X 0,Y 375.362,Z 244.126,A -85,B 0,C 180,E1 -12179.131,E2 -12179.131} C_VEL
LIN {X 0,Y 375.43,Z 241.934,A -85,B 0,C 180,E1 -12181.612,E2 -12181.612} C_VEL
LIN {X 0,Y 375.765,Z 241.678,A -85,B 0,C 180,E1 -12184.62,E2 -12184.62} C_VEL
LIN {X 0,Y 375.917,Z 241.658,A -85,B 0,C 180,E1 -12186.745,E2 -12186.745} C_VEL
LIN {X 0,Y 375.989,Z 241.651,A -85,B 0,C 180,E1 -12189.97,E2 -12189.97} C_VEL
LIN {X 0,Y 375.931,Z 241.657,A -85,B 0,C 180,E1 -12193.766,E2 -12193.766} C_VEL
LIN {X 0,Y 375.936,Z 241.654,A -85,B 0,C 180,E1 -12196.811,E2 -12196.811} C_VEL
LIN {X 0,Y 375.962,Z 241.651,A -85,B 0,C 180,E1 -12200.537,E2 -12200.537} C_VEL
LIN {X 0,Y 375.965,Z 241.654,A -85,B 0,C 180,E1 -12203.496,E2 -12203.496} C_VEL
LIN {X 0,Y 375.962,Z 241.654,A -85,B 0,C 180,E1 -12205.889,E2 -12205.889} C_VEL
LIN {X 0,Y 375.964,Z 241.655,A -85,B 0,C 180,E1 -12209.687,E2 -12209.687} C_VEL
LIN {X 0,Y 375.931,Z 241.655,A -85,B 0,C 180,E1 -12212.136,E2 -12212.136} C_VEL
LIN {X 0,Y 375.975,Z 241.651,A -85,B 0,C 180,E1 -12215.717,E2 -12215.717} C_VEL
LIN {X 0,Y 376,Z 241.652,A -85,B 0,C 180,E1 -12219.198,E2 -12219.198} C_VEL
LIN {X 0,Y 376.034,Z 241.643,A -85,B 0,C 180,E1 -12222.6,E2 -12222.6} C_VEL
LIN {X 0,Y 376.092,Z 241.635,A -85,B 0,C 180,E1 -12226.342,E2 -12226.342} C_VEL
LIN {X 0,Y 376.122,Z 241.632,A -85,B 0,C 180,E1 -12230.319,E2 -12230.319} C_VEL
LIN {X 0,Y 376.232,Z 241.62,A -85,B 0,C 180,E1 -12232.486,E2 -12232.486} C_VEL
LIN {X 0,Y 376.169,Z 241.63,A -85,B 0,C 180,E1 -12234.64,E2 -12234.64} C_VEL
LIN {X 0,Y 376.344,Z 241.603,A -85,B 0,C 180,E1 -12237.86,E2 -12237.86} C_VEL
LIN {X 0,Y 376.354,Z 241.604,A -85,B 0,C 180,E1 -12242.14,E2 -12242.14} C_VEL
LIN {X 0,Y 376.232,Z 241.623,A -85,B 0,C 180,E1 -12246.435,E2 -12246.435} C_VEL
LIN {X 0,Y 376.112,Z 241.633,A -85,B 0,C 180,E1 -12249.682,E2 -12249.682} C_VEL
LIN {X 0,Y 376.091,Z 241.636,A -85,B 0,C 180,E1 -12253.657,E2 -12253.657} C_VEL
LIN {X 0,Y 376.047,Z 241.642,A -85,B 0,C 180,E1 -12257.607,E2 -12257.607} C_VEL
LIN {X 0,Y 375.98,Z 241.648,A -85,B 0,C 180,E1 -12260.832,E2 -12260.832} C_VEL
LIN {X 0,Y 375.937,Z 241.655,A -85,B 0,C 180,E1 -12264.285,E2 -12264.285} C_VEL
LIN {X 0,Y 375.921,Z 241.655,A -85,B 0,C 180,E1 -12266.66,E2 -12266.66} C_VEL
LIN {X 0,Y 375.918,Z 241.657,A -85,B 0,C 180,E1 -12269.084,E2 -12269.084} C_VEL
LIN {X 0,Y 375.959,Z 241.657,A -85,B 0,C 180,E1 -12271.562,E2 -12271.562} C_VEL
LIN {X 0,Y 375.959,Z 241.657,A -85,B 0,C 180,E1 -12275.415,E2 -12275.415} C_VEL
LIN {X 0,Y 375.937,Z 241.653,A -85,B 0,C 180,E1 -12278.263,E2 -12278.263} C_VEL
LIN {X 0,Y 375.918,Z 241.66,A -85,B 0,C 180,E1 -12281.598,E2 -12281.598} C_VEL
LIN {X 0,Y 375.98,Z 241.677,A -85,B 0,C 180,E1 -12284.739,E2 -12284.739} C_VEL
LIN {X 0,Y 377.041,Z 247.414,A -85,B 0,C 180,E1 -12288.21,E2 -12288.21} C_VEL
LIN {X 0,Y 378.005,Z 252.949,A -85,B 0,C 180,E1 -12291.341,E2 -12291.341} C_VEL
LIN {X 0,Y 378.483,Z 257.127,A -85,B 0,C 180,E1 -12293.544,E2 -12293.544} C_VEL
LIN {X 0,Y 378.103,Z 262.318,A -85,B 0,C 180,E1 -12296.108,E2 -12296.108} C_VEL
LIN {X 0,Y 377.494,Z 268.204,A -85,B 0,C 180,E1 -12298.916,E2 -12298.916} C_VEL
LIN {X 0,Y 376.871,Z 275.311,A -85,B 0,C 180,E1 -12302.212,E2 -12302.212} C_VEL
LIN {X 0,Y 376.12,Z 284.247,A -85,B 0,C 180,E1 -12306.29,E2 -12306.29} C_VEL
LIN {X 0,Y 375.603,Z 291.976,A -85,B 0,C 180,E1 -12309.799,E2 -12309.799} C_VEL
LIN {X 0,Y 375.475,Z 293.964,A -85,B 0,C 180,E1 -12310.702,E2 -12310.702} C_VEL
LIN {X 0,Y 377.744,Z 307.437,A -85,B 0,C 180,E1 -12311.263,E2 -12311.263} C_VEL
LIN {X 0,Y 379.36,Z 319.583,A -85,B 0,C 180,E1 -12311.955,E2 -12311.955} C_VEL
LIN {X 0,Y 380.394,Z 328.651,A -85,B 0,C 180,E1 -12312.596,E2 -12312.596} C_VEL
LIN {X 0,Y 379.505,Z 339.568,A -85,B 0,C 180,E1 -12313.457,E2 -12313.457} C_VEL
LIN {X 0,Y 378.392,Z 351.405,A -85,B 0,C 180,E1 -12314.653,E2 -12314.653} C_VEL
LIN {X 0,Y 377.468,Z 361.936,A -85,B 0,C 180,E1 -12315.993,E2 -12315.993} C_VEL
LIN {X 0,Y 376.699,Z 370.466,A -85,B 0,C 180,E1 -12317.337,E2 -12317.337} C_VEL
LIN {X 0,Y 375.833,Z 378.79,A -85,B 0,C 180,E1 -12318.95,E2 -12318.95} C_VEL
LIN {X 0,Y 375.286,Z 385.512,A -85,B 0,C 180,E1 -12320.569,E2 -12320.569} C_VEL
LIN {X 0,Y 374.88,Z 391.673,A -85,B 0,C 180,E1 -12322.459,E2 -12322.459} C_VEL
LIN {X 0,Y 374.706,Z 394.958,A -85,B 0,C 180,E1 -12323.759,E2 -12323.759} C_VEL
LIN {X 0,Y 374.588,Z 398.645,A -85,B 0,C 180,E1 -12325.696,E2 -12325.696} C_VEL
LIN {X 0,Y 374.606,Z 401.068,A -85,B 0,C 180,E1 -12327.85,E2 -12327.85} C_VEL
LIN {X 0,Y 374.61,Z 401.684,A -85,B 0,C 180,E1 -12328.925,E2 -12328.925} C_VEL
LIN {X 0,Y 374.604,Z 401.902,A -85,B 0,C 180,E1 -12330,E2 -12330} C_VEL
LIN {X 0,Y 374.61,Z 401.683,A -85,B 0,C 180,E1 -12331.075,E2 -12331.075} C_VEL
LIN {X 0,Y 374.606,Z 401.068,A -85,B 0,C 180,E1 -12332.151,E2 -12332.151} C_VEL
LIN {X 0,Y 374.588,Z 398.644,A -85,B 0,C 180,E1 -12334.304,E2 -12334.304} C_VEL
LIN {X 0,Y 374.699,Z 394.973,A -85,B 0,C 180,E1 -12336.232,E2 -12336.232} C_VEL
LIN {X 0,Y 374.944,Z 390.054,A -85,B 0,C 180,E1 -12338.082,E2 -12338.082} C_VEL
LIN {X 0,Y 375.397,Z 384.483,A -85,B 0,C 180,E1 -12339.7,E2 -12339.7} C_VEL
LIN {X 0,Y 375.964,Z 377.531,A -85,B 0,C 180,E1 -12341.32,E2 -12341.32} C_VEL
LIN {X 0,Y 376.851,Z 368.851,A -85,B 0,C 180,E1 -12342.932,E2 -12342.932} C_VEL
LIN {X 0,Y 377.812,Z 359.286,A -85,B 0,C 180,E1 -12344.363,E2 -12344.363} C_VEL
LIN {X 0,Y 378.611,Z 349.008,A -85,B 0,C 180,E1 -12345.614,E2 -12345.614} C_VEL
LIN {X 0,Y 379.638,Z 337.982,A -85,B 0,C 180,E1 -12346.675,E2 -12346.675} C_VEL
LIN {X 0,Y 380.39,Z 328.598,A -85,B 0,C 180,E1 -12347.404,E2 -12347.404} C_VEL
LIN {X 0,Y 379.035,Z 316.725,A -85,B 0,C 180,E1 -12348.217,E2 -12348.217} C_VEL
LIN {X 0,Y 377.155,Z 303.517,A -85,B 0,C 180,E1 -12348.913,E2 -12348.913} C_VEL
LIN {X 0,Y 375.497,Z 293.892,A -85,B 0,C 180,E1 -12349.297,E2 -12349.297} C_VEL
LIN {X 0,Y 375.962,Z 286.832,A -85,B 0,C 180,E1 -12352.533,E2 -12352.533} C_VEL
LIN {X 0,Y 376.63,Z 277.864,A -85,B 0,C 180,E1 -12356.606,E2 -12356.606} C_VEL
LIN {X 0,Y 377.292,Z 270.053,A -85,B 0,C 180,E1 -12360.195,E2 -12360.195} C_VEL
LIN {X 0,Y 377.944,Z 263.662,A -85,B 0,C 180,E1 -12363.197,E2 -12363.197} C_VEL
LIN {X 0,Y 378.455,Z 258.315,A -85,B 0,C 180,E1 -12365.8,E2 -12365.8} C_VEL
LIN {X 0,Y 378.262,Z 254.434,A -85,B 0,C 180,E1 -12367.817,E2 -12367.817} C_VEL
LIN {X 0,Y 377.385,Z 249.303,A -85,B 0,C 180,E1 -12370.678,E2 -12370.678} C_VEL
LIN {X 0,Y 376.424,Z 244.182,A -85,B 0,C 180,E1 -12373.695,E2 -12373.695} C_VEL
LIN {X 0,Y 375.983,Z 241.657,A -85,B 0,C 180,E1 -12375.261,E2 -12375.261} C_VEL
LIN {X 0,Y 375.918,Z 241.658,A -85,B 0,C 180,E1 -12379.13,E2 -12379.13} C_VEL
LIN {X 0,Y 375.956,Z 241.651,A -85,B 0,C 180,E1 -12381.91,E2 -12381.91} C_VEL
LIN {X 0,Y 375.983,Z 241.648,A -85,B 0,C 180,E1 -12385.333,E2 -12385.333} C_VEL
LIN {X 0,Y 375.961,Z 241.657,A -85,B 0,C 180,E1 -12388.438,E2 -12388.438} C_VEL
LIN {X 0,Y 375.929,Z 241.659,A -85,B 0,C 180,E1 -12392.136,E2 -12392.136} C_VEL
LIN {X 0,Y 375.939,Z 241.656,A -85,B 0,C 180,E1 -12394.534,E2 -12394.534} C_VEL
LIN {X 0,Y 375.978,Z 241.649,A -85,B 0,C 180,E1 -12396.887,E2 -12396.887} C_VEL
LIN {X 0,Y 376.002,Z 241.649,A -85,B 0,C 180,E1 -12400.34,E2 -12400.34} C_VEL
LIN {X 0,Y 376.033,Z 241.645,A -85,B 0,C 180,E1 -12403.719,E2 -12403.719} C_VEL
LIN {X 0,Y 376.106,Z 241.632,A -85,B 0,C 180,E1 -12407.042,E2 -12407.042} C_VEL
LIN {X 0,Y 376.112,Z 241.633,A -85,B 0,C 180,E1 -12410.318,E2 -12410.318} C_VEL
LIN {X 0,Y 376.234,Z 241.622,A -85,B 0,C 180,E1 -12413.565,E2 -12413.565} C_VEL
LIN {X 0,Y 376.356,Z 241.604,A -85,B 0,C 180,E1 -12417.86,E2 -12417.86} C_VEL
LIN {X 0,Y 376.346,Z 241.603,A -85,B 0,C 180,E1 -12422.14,E2 -12422.14} C_VEL
LIN {X 0,Y 376.216,Z 241.618,A -85,B 0,C 180,E1 -12426.614,E2 -12426.614} C_VEL
LIN {X 0,Y 376.118,Z 241.633,A -85,B 0,C 180,E1 -12429.682,E2 -12429.682} C_VEL
LIN {X 0,Y 376.094,Z 241.635,A -85,B 0,C 180,E1 -12433.658,E2 -12433.658} C_VEL
LIN {X 0,Y 376.031,Z 241.642,A -85,B 0,C 180,E1 -12437.599,E2 -12437.599} C_VEL
LIN {X 0,Y 375.982,Z 241.654,A -85,B 0,C 180,E1 -12440.832,E2 -12440.832} C_VEL
LIN {X 0,Y 375.979,Z 241.65,A -85,B 0,C 180,E1 -12444.283,E2 -12444.283} C_VEL
LIN {X 0,Y 375.933,Z 241.654,A -85,B 0,C 180,E1 -12447.864,E2 -12447.864} C_VEL
LIN {X 0,Y 375.96,Z 241.65,A -85,B 0,C 180,E1 -12451.562,E2 -12451.562} C_VEL
LIN {X 0,Y 375.961,Z 241.65,A -85,B 0,C 180,E1 -12455.415,E2 -12455.415} C_VEL
LIN {X 0,Y 375.975,Z 241.655,A -85,B 0,C 180,E1 -12458.27,E2 -12458.27} C_VEL
LIN {X 0,Y 375.936,Z 241.655,A -85,B 0,C 180,E1 -12461.6,E2 -12461.6} C_VEL
LIN {X 0,Y 375.93,Z 241.654,A -85,B 0,C 180,E1 -12465.269,E2 -12465.269} C_VEL
LIN {X 0,Y 375.929,Z 241.657,A -85,B 0,C 180,E1 -12468.401,E2 -12468.401} C_VEL
LIN {X 0,Y 375.972,Z 241.654,A -85,B 0,C 180,E1 -12471.73,E2 -12471.73} C_VEL
LIN {X 0,Y 375.844,Z 241.665,A -85,B 0,C 180,E1 -12474.572,E2 -12474.572} C_VEL
LIN {X 0,Y 375.547,Z 241.708,A -85,B 0,C 180,E1 -12477.366,E2 -12477.366} C_VEL
LIN {X 0,Y 375.424,Z 241.826,A -85,B 0,C 180,E1 -12478.388,E2 -12478.388} C_VEL
LIN {X 0,Y 375.357,Z 245.114,A -85,B 0,C 180,E1 -12482.089,E2 -12482.089} C_VEL
LIN {X 0,Y 375.203,Z 248.469,A -85,B 0,C 180,E1 -12485.664,E2 -12485.664} C_VEL
LIN {X 0,Y 375.156,Z 251.953,A -85,B 0,C 180,E1 -12489.149,E2 -12489.149} C_VEL
LIN {X 0,Y 375.125,Z 253.664,A -85,B 0,C 180,E1 -12490.79,E2 -12490.79} C_VEL
LIN {X 0,Y 379.129,Z 268.043,A -85,B 0,C 180,E1 -12491.561,E2 -12491.561} C_VEL
LIN {X 0,Y 381.657,Z 279.362,A -85,B 0,C 180,E1 -12492.329,E2 -12492.329} C_VEL
LIN {X 0,Y 381.008,Z 290.4,A -85,B 0,C 180,E1 -12493.111,E2 -12493.111} C_VEL
LIN {X 0,Y 380.167,Z 301.2,A -85,B 0,C 180,E1 -12494.088,E2 -12494.088} C_VEL
LIN {X 0,Y 379.298,Z 311.38,A -85,B 0,C 180,E1 -12495.24,E2 -12495.24} C_VEL
LIN {X 0,Y 378.342,Z 320.953,A -85,B 0,C 180,E1 -12496.573,E2 -12496.573} C_VEL
LIN {X 0,Y 377.54,Z 328.788,A -85,B 0,C 180,E1 -12497.911,E2 -12497.911} C_VEL
LIN {X 0,Y 376.731,Z 336.441,A -85,B 0,C 180,E1 -12499.52,E2 -12499.52} C_VEL
LIN {X 0,Y 376.132,Z 341.663,A -85,B 0,C 180,E1 -12500.861,E2 -12500.861} C_VEL
LIN {X 0,Y 375.609,Z 347.07,A -85,B 0,C 180,E1 -12502.606,E2 -12502.606} C_VEL
LIN {X 0,Y 375.095,Z 351.71,A -85,B 0,C 180,E1 -12504.624,E2 -12504.624} C_VEL
LIN {X 0,Y 375.065,Z 353.548,A -85,B 0,C 180,E1 -12505.701,E2 -12505.701} C_VEL
LIN {X 0,Y 374.986,Z 354.935,A -85,B 0,C 180,E1 -12506.777,E2 -12506.777} C_VEL
LIN {X 0,Y 374.707,Z 356.54,A -85,B 0,C 180,E1 -12508.925,E2 -12508.925} C_VEL
LIN {X 0,Y 374.687,Z 356.772,A -85,B 0,C 180,E1 -12510,E2 -12510} C_VEL
LIN {X 0,Y 374.807,Z 356,A -85,B 0,C 180,E1 -12512.149,E2 -12512.149} C_VEL
LIN {X 0,Y 374.98,Z 355.035,A -85,B 0,C 180,E1 -12513.223,E2 -12513.223} C_VEL
LIN {X 0,Y 375.057,Z 353.691,A -85,B 0,C 180,E1 -12514.298,E2 -12514.298} C_VEL
LIN {X 0,Y 375.2,Z 350.852,A -85,B 0,C 180,E1 -12515.913,E2 -12515.913} C_VEL
LIN {X 0,Y 375.595,Z 346.99,A -85,B 0,C 180,E1 -12517.526,E2 -12517.526} C_VEL
LIN {X 0,Y 376.08,Z 342.007,A -85,B 0,C 180,E1 -12519.14,E2 -12519.14} C_VEL
LIN {X 0,Y 376.8,Z 335.724,A -85,B 0,C 180,E1 -12520.75,E2 -12520.75} C_VEL
LIN {X 0,Y 377.634,Z 327.859,A -85,B 0,C 180,E1 -12522.358,E2 -12522.358} C_VEL
LIN {X 0,Y 378.693,Z 318.065,A -85,B 0,C 180,E1 -12523.961,E2 -12523.961} C_VEL
LIN {X 0,Y 379.61,Z 308.621,A -85,B 0,C 180,E1 -12525.198,E2 -12525.198} C_VEL
LIN {X 0,Y 380.483,Z 297.59,A -85,B 0,C 180,E1 -12526.361,E2 -12526.361} C_VEL
LIN {X 0,Y 381.397,Z 285.65,A -85,B 0,C 180,E1 -12527.347,E2 -12527.347} C_VEL
LIN {X 0,Y 381.593,Z 278.676,A -85,B 0,C 180,E1 -12527.818,E2 -12527.818} C_VEL
LIN {X 0,Y 378.723,Z 266.356,A -85,B 0,C 180,E1 -12528.64,E2 -12528.64} C_VEL
LIN {X 0,Y 375.122,Z 253.61,A -85,B 0,C 180,E1 -12529.326,E2 -12529.326} C_VEL
LIN {X 0,Y 375.175,Z 250.08,A -85,B 0,C 180,E1 -12532.798,E2 -12532.798} C_VEL
LIN {X 0,Y 374.558,Z 249.294,A -85,B 0,C 180,E1 -12533.686,E2 -12533.686} C_VEL
LIN {X 0,Y 371.737,Z 248.252,A -85,B 0,C 180,E1 -12535.137,E2 -12535.137} C_VEL
LIN {X 0,Y 369.329,Z 247.452,A -85,B 0,C 180,E1 -12536.31,E2 -12536.31} C_VEL
LIN {X 0,Y 368.306,Z 246.745,A -85,B 0,C 180,E1 -12537.215,E2 -12537.215} C_VEL
LIN {X 0,Y 368.229,Z 246.474,A -85,B 0,C 180,E1 -12537.521,E2 -12537.521} C_VEL
LIN {X 0,Y 368.365,Z 243.372,A -85,B 0,C 180,E1 -12541.006,E2 -12541.006} C_VEL
LIN {X 0,Y 368.439,Z 242.594,A -85,B 0,C 180,E1 -12542.283,E2 -12542.283} C_VEL
LIN {X 0,Y 368.763,Z 242.548,A -85,B 0,C 180,E1 -12544.964,E2 -12544.964} C_VEL
LIN {X 0,Y 368.874,Z 242.534,A -85,B 0,C 180,E1 -12547.567,E2 -12547.567} C_VEL
LIN {X 0,Y 368.911,Z 242.532,A -85,B 0,C 180,E1 -12550.37,E2 -12550.37} C_VEL
LIN {X 0,Y 368.884,Z 242.534,A -85,B 0,C 180,E1 -12553.616,E2 -12553.616} C_VEL
LIN {X 0,Y 368.887,Z 242.532,A -85,B 0,C 180,E1 -12556.696,E2 -12556.696} C_VEL
LIN {X 0,Y 368.912,Z 242.532,A -85,B 0,C 180,E1 -12559.643,E2 -12559.643} C_VEL
LIN {X 0,Y 368.902,Z 242.531,A -85,B 0,C 180,E1 -12563.144,E2 -12563.144} C_VEL
LIN {X 0,Y 368.9,Z 242.53,A -85,B 0,C 180,E1 -12566.462,E2 -12566.462} C_VEL
LIN {X 0,Y 368.931,Z 242.527,A -85,B 0,C 180,E1 -12569.046,E2 -12569.046} C_VEL
LIN {X 0,Y 368.87,Z 242.534,A -85,B 0,C 180,E1 -12572.789,E2 -12572.789} C_VEL
LIN {X 0,Y 368.951,Z 242.523,A -85,B 0,C 180,E1 -12576.42,E2 -12576.42} C_VEL
LIN {X 0,Y 368.938,Z 242.526,A -85,B 0,C 180,E1 -12579.947,E2 -12579.947} C_VEL
LIN {X 0,Y 368.969,Z 242.524,A -85,B 0,C 180,E1 -12583.398,E2 -12583.398} C_VEL
LIN {X 0,Y 369.06,Z 242.514,A -85,B 0,C 180,E1 -12586.79,E2 -12586.79} C_VEL
LIN {X 0,Y 369.07,Z 242.509,A -85,B 0,C 180,E1 -12590.132,E2 -12590.132} C_VEL
LIN {X 0,Y 369.19,Z 242.495,A -85,B 0,C 180,E1 -12592.342,E2 -12592.342} C_VEL
LIN {X 0,Y 369.142,Z 242.504,A -85,B 0,C 180,E1 -12594.537,E2 -12594.537} C_VEL
LIN {X 0,Y 369.308,Z 242.479,A -85,B 0,C 180,E1 -12597.819,E2 -12597.819} C_VEL
LIN {X 0,Y 369.319,Z 242.481,A -85,B 0,C 180,E1 -12602.181,E2 -12602.181} C_VEL
LIN {X 0,Y 369.19,Z 242.498,A -85,B 0,C 180,E1 -12606.558,E2 -12606.558} C_VEL
LIN {X 0,Y 369.062,Z 242.512,A -85,B 0,C 180,E1 -12609.868,E2 -12609.868} C_VEL
LIN {X 0,Y 369.039,Z 242.515,A -85,B 0,C 180,E1 -12613.772,E2 -12613.772} C_VEL
LIN {X 0,Y 369.003,Z 242.521,A -85,B 0,C 180,E1 -12617.768,E2 -12617.768} C_VEL
LIN {X 0,Y 368.911,Z 242.529,A -85,B 0,C 180,E1 -12621.221,E2 -12621.221} C_VEL
LIN {X 0,Y 368.912,Z 242.534,A -85,B 0,C 180,E1 -12623.875,E2 -12623.875} C_VEL
LIN {X 0,Y 368.866,Z 242.536,A -85,B 0,C 180,E1 -12627.211,E2 -12627.211} C_VEL
LIN {X 0,Y 368.931,Z 242.527,A -85,B 0,C 180,E1 -12630.953,E2 -12630.953} C_VEL
LIN {X 0,Y 368.93,Z 242.528,A -85,B 0,C 180,E1 -12635.001,E2 -12635.001} C_VEL
LIN {X 0,Y 368.878,Z 242.533,A -85,B 0,C 180,E1 -12638.634,E2 -12638.634} C_VEL
LIN {X 0,Y 368.871,Z 242.537,A -85,B 0,C 180,E1 -12642.007,E2 -12642.007} C_VEL
LIN {X 0,Y 368.927,Z 242.603,A -85,B 0,C 180,E1 -12644.328,E2 -12644.328} C_VEL
LIN {X 0,Y 369.97,Z 248.174,A -85,B 0,C 180,E1 -12647.804,E2 -12647.804} C_VEL
LIN {X 0,Y 371.028,Z 254.247,A -85,B 0,C 180,E1 -12651.311,E2 -12651.311} C_VEL
LIN {X 0,Y 371.48,Z 258.128,A -85,B 0,C 180,E1 -12653.42,E2 -12653.42} C_VEL
LIN {X 0,Y 371.112,Z 263.22,A -85,B 0,C 180,E1 -12655.983,E2 -12655.983} C_VEL
LIN {X 0,Y 370.38,Z 269.776,A -85,B 0,C 180,E1 -12659.181,E2 -12659.181} C_VEL
LIN {X 0,Y 369.805,Z 276.257,A -85,B 0,C 180,E1 -12662.25,E2 -12662.25} C_VEL
LIN {X 0,Y 369.073,Z 284.421,A -85,B 0,C 180,E1 -12666.069,E2 -12666.069} C_VEL
LIN {X 0,Y 368.634,Z 290.921,A -85,B 0,C 180,E1 -12669.097,E2 -12669.097} C_VEL
LIN {X 0,Y 368.453,Z 293.545,A -85,B 0,C 180,E1 -12670.32,E2 -12670.32} C_VEL
LIN {X 0,Y 370.858,Z 307.327,A -85,B 0,C 180,E1 -12670.916,E2 -12670.916} C_VEL
LIN {X 0,Y 372.467,Z 319.914,A -85,B 0,C 180,E1 -12671.657,E2 -12671.657} C_VEL
LIN {X 0,Y 373.49,Z 329.682,A -85,B 0,C 180,E1 -12672.376,E2 -12672.376} C_VEL
LIN {X 0,Y 372.406,Z 342.008,A -85,B 0,C 180,E1 -12673.415,E2 -12673.415} C_VEL
LIN {X 0,Y 371.282,Z 353.3,A -85,B 0,C 180,E1 -12674.633,E2 -12674.633} C_VEL
LIN {X 0,Y 370.351,Z 363.315,A -85,B 0,C 180,E1 -12675.998,E2 -12675.998} C_VEL
LIN {X 0,Y 369.437,Z 373.036,A -85,B 0,C 180,E1 -12677.642,E2 -12677.642} C_VEL
LIN {X 0,Y 368.616,Z 380.776,A -85,B 0,C 180,E1 -12679.287,E2 -12679.287} C_VEL
LIN {X 0,Y 368.036,Z 387.927,A -85,B 0,C 180,E1 -12681.213,E2 -12681.213} C_VEL
LIN {X 0,Y 367.747,Z 392.692,A -85,B 0,C 180,E1 -12682.864,E2 -12682.864} C_VEL
LIN {X 0,Y 367.563,Z 396.336,A -85,B 0,C 180,E1 -12684.514,E2 -12684.514} C_VEL
LIN {X 0,Y 367.519,Z 398.218,A -85,B 0,C 180,E1 -12685.613,E2 -12685.613} C_VEL
LIN {X 0,Y 367.51,Z 400.641,A -85,B 0,C 180,E1 -12687.808,E2 -12687.808} C_VEL
LIN {X 0,Y 367.546,Z 401.258,A -85,B 0,C 180,E1 -12688.905,E2 -12688.905} C_VEL
LIN {X 0,Y 367.538,Z 401.477,A -85,B 0,C 180,E1 -12690,E2 -12690} C_VEL
LIN {X 0,Y 367.546,Z 401.258,A -85,B 0,C 180,E1 -12691.096,E2 -12691.096} C_VEL
LIN {X 0,Y 367.51,Z 400.64,A -85,B 0,C 180,E1 -12692.192,E2 -12692.192} C_VEL
LIN {X 0,Y 367.518,Z 398.217,A -85,B 0,C 180,E1 -12694.387,E2 -12694.387} C_VEL
LIN {X 0,Y 367.598,Z 394.923,A -85,B 0,C 180,E1 -12696.187,E2 -12696.187} C_VEL
LIN {X 0,Y 367.893,Z 389.624,A -85,B 0,C 180,E1 -12698.238,E2 -12698.238} C_VEL
LIN {X 0,Y 368.344,Z 384.05,A -85,B 0,C 180,E1 -12699.888,E2 -12699.888} C_VEL
LIN {X 0,Y 368.944,Z 377.098,A -85,B 0,C 180,E1 -12701.538,E2 -12701.538} C_VEL
LIN {X 0,Y 369.878,Z 368.418,A -85,B 0,C 180,E1 -12703.18,E2 -12703.18} C_VEL
LIN {X 0,Y 370.82,Z 359.712,A -85,B 0,C 180,E1 -12704.517,E2 -12704.517} C_VEL
LIN {X 0,Y 371.623,Z 349.758,A -85,B 0,C 180,E1 -12705.775,E2 -12705.775} C_VEL
LIN {X 0,Y 372.664,Z 339.095,A -85,B 0,C 180,E1 -12706.856,E2 -12706.856} C_VEL
LIN {X 0,Y 373.47,Z 328.298,A -85,B 0,C 180,E1 -12707.727,E2 -12707.727} C_VEL
LIN {X 0,Y 372.088,Z 316.277,A -85,B 0,C 180,E1 -12708.57,E2 -12708.57} C_VEL
LIN {X 0,Y 370.093,Z 302.642,A -85,B 0,C 180,E1 -12709.304,E2 -12709.304} C_VEL
LIN {X 0,Y 368.455,Z 293.493,A -85,B 0,C 180,E1 -12709.681,E2 -12709.681} C_VEL
LIN {X 0,Y 368.948,Z 286.44,A -85,B 0,C 180,E1 -12712.986,E2 -12712.986} C_VEL
LIN {X 0,Y 369.597,Z 278.559,A -85,B 0,C 180,E1 -12716.655,E2 -12716.655} C_VEL
LIN {X 0,Y 370.252,Z 271.023,A -85,B 0,C 180,E1 -12720.2,E2 -12720.2} C_VEL
LIN {X 0,Y 370.996,Z 264.103,A -85,B 0,C 180,E1 -12723.538,E2 -12723.538} C_VEL
LIN {X 0,Y 371.486,Z 259.358,A -85,B 0,C 180,E1 -12725.908,E2 -12725.908} C_VEL
LIN {X 0,Y 371.233,Z 255.478,A -85,B 0,C 180,E1 -12727.972,E2 -12727.972} C_VEL
LIN {X 0,Y 370.154,Z 249.061,A -85,B 0,C 180,E1 -12731.647,E2 -12731.647} C_VEL
LIN {X 0,Y 369.065,Z 243.307,A -85,B 0,C 180,E1 -12735.204,E2 -12735.204} C_VEL
LIN {X 0,Y 368.9,Z 242.534,A -85,B 0,C 180,E1 -12735.831,E2 -12735.831} C_VEL
LIN {X 0,Y 368.886,Z 242.532,A -85,B 0,C 180,E1 -12739.648,E2 -12739.648} C_VEL
LIN {X 0,Y 368.902,Z 242.531,A -85,B 0,C 180,E1 -12743.145,E2 -12743.145} C_VEL
LIN {X 0,Y 368.9,Z 242.536,A -85,B 0,C 180,E1 -12746.462,E2 -12746.462} C_VEL
LIN {X 0,Y 368.933,Z 242.527,A -85,B 0,C 180,E1 -12749.047,E2 -12749.047} C_VEL
LIN {X 0,Y 368.868,Z 242.536,A -85,B 0,C 180,E1 -12752.789,E2 -12752.789} C_VEL
LIN {X 0,Y 368.949,Z 242.528,A -85,B 0,C 180,E1 -12756.42,E2 -12756.42} C_VEL
LIN {X 0,Y 368.941,Z 242.53,A -85,B 0,C 180,E1 -12759.947,E2 -12759.947} C_VEL
LIN {X 0,Y 368.98,Z 242.521,A -85,B 0,C 180,E1 -12763.399,E2 -12763.399} C_VEL
LIN {X 0,Y 369.061,Z 242.51,A -85,B 0,C 180,E1 -12766.79,E2 -12766.79} C_VEL
LIN {X 0,Y 369.063,Z 242.512,A -85,B 0,C 180,E1 -12770.132,E2 -12770.132} C_VEL
LIN {X 0,Y 369.192,Z 242.497,A -85,B 0,C 180,E1 -12773.442,E2 -12773.442} C_VEL
LIN {X 0,Y 369.321,Z 242.481,A -85,B 0,C 180,E1 -12777.819,E2 -12777.819} C_VEL
LIN {X 0,Y 369.31,Z 242.479,A -85,B 0,C 180,E1 -12782.181,E2 -12782.181} C_VEL
LIN {X 0,Y 369.188,Z 242.494,A -85,B 0,C 180,E1 -12786.597,E2 -12786.597} C_VEL
LIN {X 0,Y 369.068,Z 242.509,A -85,B 0,C 180,E1 -12789.868,E2 -12789.868} C_VEL
LIN {X 0,Y 369.042,Z 242.513,A -85,B 0,C 180,E1 -12793.772,E2 -12793.772} C_VEL
LIN {X 0,Y 368.995,Z 242.518,A -85,B 0,C 180,E1 -12797.743,E2 -12797.743} C_VEL
LIN {X 0,Y 368.914,Z 242.53,A -85,B 0,C 180,E1 -12801.221,E2 -12801.221} C_VEL
LIN {X 0,Y 368.934,Z 242.531,A -85,B 0,C 180,E1 -12804.777,E2 -12804.777} C_VEL
LIN {X 0,Y 368.916,Z 242.533,A -85,B 0,C 180,E1 -12808.442,E2 -12808.442} C_VEL
LIN {X 0,Y 368.901,Z 242.533,A -85,B 0,C 180,E1 -12812.238,E2 -12812.238} C_VEL
LIN {X 0,Y 368.932,Z 242.527,A -85,B 0,C 180,E1 -12815.001,E2 -12815.001} C_VEL
LIN {X 0,Y 368.909,Z 242.531,A -85,B 0,C 180,E1 -12818.64,E2 -12818.64} C_VEL
LIN {X 0,Y 368.884,Z 242.536,A -85,B 0,C 180,E1 -12822.009,E2 -12822.009} C_VEL
LIN {X 0,Y 368.883,Z 242.532,A -85,B 0,C 180,E1 -12825.176,E2 -12825.176} C_VEL
LIN {X 0,Y 368.879,Z 242.537,A -85,B 0,C 180,E1 -12828.177,E2 -12828.177} C_VEL
LIN {X 0,Y 368.907,Z 242.53,A -85,B 0,C 180,E1 -12831.361,E2 -12831.361} C_VEL
LIN {X 0,Y 368.856,Z 242.542,A -85,B 0,C 180,E1 -12833.796,E2 -12833.796} C_VEL
LIN {X 0,Y 368.529,Z 242.581,A -85,B 0,C 180,E1 -12837.045,E2 -12837.045} C_VEL
LIN {X 0,Y 368.44,Z 242.593,A -85,B 0,C 180,E1 -12837.717,E2 -12837.717} C_VEL
LIN {X 0,Y 368.354,Z 243.422,A -85,B 0,C 180,E1 -12839.158,E2 -12839.158} C_VEL
LIN {X 0,Y 368.253,Z 246.596,A -85,B 0,C 180,E1 -12842.739,E2 -12842.739} C_VEL
LIN {X 0,Y 368.158,Z 250.02,A -85,B 0,C 180,E1 -12846.392,E2 -12846.392} C_VEL
LIN {X 0,Y 368.097,Z 254.07,A -85,B 0,C 180,E1 -12850.379,E2 -12850.379} C_VEL
LIN {X 0,Y 368.62,Z 256.193,A -85,B 0,C 180,E1 -12850.512,E2 -12850.512} C_VEL
LIN {X 0,Y 372.372,Z 269.216,A -85,B 0,C 180,E1 -12851.249,E2 -12851.249} C_VEL
LIN {X 0,Y 374.816,Z 280.259,A -85,B 0,C 180,E1 -12852.024,E2 -12852.024} C_VEL
LIN {X 0,Y 374.135,Z 292.414,A -85,B 0,C 180,E1 -12852.931,E2 -12852.931} C_VEL
LIN {X 0,Y 373.23,Z 303.813,A -85,B 0,C 180,E1 -12854.023,E2 -12854.023} C_VEL
LIN {X 0,Y 372.304,Z 313.924,A -85,B 0,C 180,E1 -12855.236,E2 -12855.236} C_VEL
LIN {X 0,Y 371.293,Z 323.069,A -85,B 0,C 180,E1 -12856.592,E2 -12856.592} C_VEL
LIN {X 0,Y 370.289,Z 331.942,A -85,B 0,C 180,E1 -12858.227,E2 -12858.227} C_VEL
LIN {X 0,Y 369.472,Z 339.08,A -85,B 0,C 180,E1 -12859.866,E2 -12859.866} C_VEL
LIN {X 0,Y 368.947,Z 343.89,A -85,B 0,C 180,E1 -12861.234,E2 -12861.234} C_VEL
LIN {X 0,Y 368.436,Z 348.971,A -85,B 0,C 180,E1 -12863.039,E2 -12863.039} C_VEL
LIN {X 0,Y 368.046,Z 352.137,A -85,B 0,C 180,E1 -12864.521,E2 -12864.521} C_VEL
LIN {X 0,Y 367.985,Z 353.977,A -85,B 0,C 180,E1 -12865.618,E2 -12865.618} C_VEL
LIN {X 0,Y 367.932,Z 355.361,A -85,B 0,C 180,E1 -12866.715,E2 -12866.715} C_VEL
LIN {X 0,Y 367.64,Z 356.966,A -85,B 0,C 180,E1 -12868.904,E2 -12868.904} C_VEL
LIN {X 0,Y 367.617,Z 357.198,A -85,B 0,C 180,E1 -12870,E2 -12870} C_VEL
LIN {X 0,Y 367.747,Z 356.425,A -85,B 0,C 180,E1 -12872.19,E2 -12872.19} C_VEL
LIN {X 0,Y 367.926,Z 355.46,A -85,B 0,C 180,E1 -12873.285,E2 -12873.285} C_VEL
LIN {X 0,Y 367.977,Z 354.118,A -85,B 0,C 180,E1 -12874.381,E2 -12874.381} C_VEL
LIN {X 0,Y 368.168,Z 351.277,A -85,B 0,C 180,E1 -12876.026,E2 -12876.026} C_VEL
LIN {X 0,Y 368.584,Z 347.414,A -85,B 0,C 180,E1 -12877.67,E2 -12877.67} C_VEL
LIN {X 0,Y 369.089,Z 342.432,A -85,B 0,C 180,E1 -12879.314,E2 -12879.314} C_VEL
LIN {X 0,Y 369.848,Z 336.148,A -85,B 0,C 180,E1 -12880.954,E2 -12880.954} C_VEL
LIN {X 0,Y 370.727,Z 328.282,A -85,B 0,C 180,E1 -12882.592,E2 -12882.592} C_VEL
LIN {X 0,Y 371.831,Z 318.488,A -85,B 0,C 180,E1 -12884.224,E2 -12884.224} C_VEL
LIN {X 0,Y 372.77,Z 309.12,A -85,B 0,C 180,E1 -12885.474,E2 -12885.474} C_VEL
LIN {X 0,Y 373.693,Z 298.011,A -85,B 0,C 180,E1 -12886.667,E2 -12886.667} C_VEL
LIN {X 0,Y 374.629,Z 286.188,A -85,B 0,C 180,E1 -12887.661,E2 -12887.661} C_VEL
LIN {X 0,Y 374.763,Z 279.608,A -85,B 0,C 180,E1 -12888.122,E2 -12888.122} C_VEL
LIN {X 0,Y 371.85,Z 267.263,A -85,B 0,C 180,E1 -12888.975,E2 -12888.975} C_VEL
LIN {X 0,Y 368.089,Z 254.036,A -85,B 0,C 180,E1 -12889.706,E2 -12889.706} C_VEL
LIN {X 0,Y 368.169,Z 250.114,A -85,B 0,C 180,E1 -12893.633,E2 -12893.633} C_VEL
LIN {X 0,Y 368.228,Z 246.712,A -85,B 0,C 180,E1 -12897.262,E2 -12897.262} C_VEL
LIN {X 0,Y 368.229,Z 246.474,A -85,B 0,C 180,E1 -12897.521,E2 -12897.521} C_VEL
LIN {X 0,Y 367.578,Z 245.742,A -85,B 0,C 180,E1 -12898.427,E2 -12898.427} C_VEL
LIN {X 0,Y 364.743,Z 244.796,A -85,B 0,C 180,E1 -12899.906,E2 -12899.906} C_VEL
LIN {X 0,Y 362.381,Z 244.072,A -85,B 0,C 180,E1 -12901.105,E2 -12901.105} C_VEL
LIN {X 0,Y 361.435,Z 243.664,A -85,B 0,C 180,E1 -12902.034,E2 -12902.034} C_VEL
LIN {X 0,Y 361.394,Z 243.584,A -85,B 0,C 180,E1 -12902.349,E2 -12902.349} C_VEL
LIN {X 0,Y 361.748,Z 243.422,A -85,B 0,C 180,E1 -12905.65,E2 -12905.65} C_VEL
LIN {X 0,Y 361.868,Z 243.406,A -85,B 0,C 180,E1 -12909.026,E2 -12909.026} C_VEL
LIN {X 0,Y 361.838,Z 243.41,A -85,B 0,C 180,E1 -12912.829,E2 -12912.829} C_VEL
LIN {X 0,Y 361.82,Z 243.418,A -85,B 0,C 180,E1 -12915.946,E2 -12915.946} C_VEL
LIN {X 0,Y 361.836,Z 243.411,A -85,B 0,C 180,E1 -12919.245,E2 -12919.245} C_VEL
LIN {X 0,Y 361.865,Z 243.406,A -85,B 0,C 180,E1 -12922.777,E2 -12922.777} C_VEL
LIN {X 0,Y 361.857,Z 243.413,A -85,B 0,C 180,E1 -12925.72,E2 -12925.72} C_VEL
LIN {X 0,Y 361.866,Z 243.411,A -85,B 0,C 180,E1 -12929.671,E2 -12929.671} C_VEL
LIN {X 0,Y 361.866,Z 243.412,A -85,B 0,C 180,E1 -12933.468,E2 -12933.468} C_VEL
LIN {X 0,Y 361.88,Z 243.409,A -85,B 0,C 180,E1 -12937.144,E2 -12937.144} C_VEL
LIN {X 0,Y 361.888,Z 243.405,A -85,B 0,C 180,E1 -12940.722,E2 -12940.722} C_VEL
LIN {X 0,Y 361.943,Z 243.397,A -85,B 0,C 180,E1 -12944.226,E2 -12944.226} C_VEL
LIN {X 0,Y 362.001,Z 243.391,A -85,B 0,C 180,E1 -12946.528,E2 -12946.528} C_VEL
LIN {X 0,Y 362.034,Z 243.385,A -85,B 0,C 180,E1 -12949.938,E2 -12949.938} C_VEL
LIN {X 0,Y 362.153,Z 243.371,A -85,B 0,C 180,E1 -12952.193,E2 -12952.193} C_VEL
LIN {X 0,Y 362.116,Z 243.378,A -85,B 0,C 180,E1 -12954.431,E2 -12954.431} C_VEL
LIN {X 0,Y 362.271,Z 243.356,A -85,B 0,C 180,E1 -12957.776,E2 -12957.776} C_VEL
LIN {X 0,Y 362.283,Z 243.358,A -85,B 0,C 180,E1 -12962.223,E2 -12962.223} C_VEL
LIN {X 0,Y 362.151,Z 243.373,A -85,B 0,C 180,E1 -12966.687,E2 -12966.687} C_VEL
LIN {X 0,Y 361.999,Z 243.394,A -85,B 0,C 180,E1 -12970.063,E2 -12970.063} C_VEL
LIN {X 0,Y 362,Z 243.393,A -85,B 0,C 180,E1 -12973.899,E2 -12973.899} C_VEL
LIN {X 0,Y 361.97,Z 243.399,A -85,B 0,C 180,E1 -12977.939,E2 -12977.939} C_VEL
LIN {X 0,Y 361.856,Z 243.411,A -85,B 0,C 180,E1 -12981.655,E2 -12981.655} C_VEL
LIN {X 0,Y 361.863,Z 243.408,A -85,B 0,C 180,E1 -12985.295,E2 -12985.295} C_VEL
LIN {X 0,Y 361.856,Z 243.409,A -85,B 0,C 180,E1 -12989.074,E2 -12989.074} C_VEL
LIN {X 0,Y 361.85,Z 243.409,A -85,B 0,C 180,E1 -12992.945,E2 -12992.945} C_VEL
LIN {X 0,Y 361.869,Z 243.41,A -85,B 0,C 180,E1 -12995.637,E2 -12995.637} C_VEL
LIN {X 0,Y 361.827,Z 243.414,A -85,B 0,C 180,E1 -12999.018,E2 -12999.018} C_VEL
LIN {X 0,Y 361.834,Z 243.416,A -85,B 0,C 180,E1 -13002.829,E2 -13002.829} C_VEL
LIN {X 0,Y 361.882,Z 243.635,A -85,B 0,C 180,E1 -13003.966,E2 -13003.966} C_VEL
LIN {X 0,Y 362.876,Z 248.945,A -85,B 0,C 180,E1 -13007.389,E2 -13007.389} C_VEL
LIN {X 0,Y 363.838,Z 254.322,A -85,B 0,C 180,E1 -13010.593,E2 -13010.593} C_VEL
LIN {X 0,Y 364.479,Z 259.146,A -85,B 0,C 180,E1 -13013.291,E2 -13013.291} C_VEL
LIN {X 0,Y 364.078,Z 264.603,A -85,B 0,C 180,E1 -13016.104,E2 -13016.104} C_VEL
LIN {X 0,Y 363.362,Z 270.752,A -85,B 0,C 180,E1 -13019.166,E2 -13019.166} C_VEL
LIN {X 0,Y 362.741,Z 277.188,A -85,B 0,C 180,E1 -13022.29,E2 -13022.29} C_VEL
LIN {X 0,Y 362.024,Z 284.801,A -85,B 0,C 180,E1 -13025.941,E2 -13025.941} C_VEL
LIN {X 0,Y 361.448,Z 292.897,A -85,B 0,C 180,E1 -13029.811,E2 -13029.811} C_VEL
LIN {X 0,Y 361.424,Z 293.125,A -85,B 0,C 180,E1 -13029.921,E2 -13029.921} C_VEL
LIN {X 0,Y 363.881,Z 307.029,A -85,B 0,C 180,E1 -13030.542,E2 -13030.542} C_VEL
LIN {X 0,Y 365.596,Z 320.229,A -85,B 0,C 180,E1 -13031.347,E2 -13031.347} C_VEL
LIN {X 0,Y 366.621,Z 330.536,A -85,B 0,C 180,E1 -13032.139,E2 -13032.139} C_VEL
LIN {X 0,Y 365.444,Z 343.01,A -85,B 0,C 180,E1 -13033.234,E2 -13033.234} C_VEL
LIN {X 0,Y 364.388,Z 352.872,A -85,B 0,C 180,E1 -13034.335,E2 -13034.335} C_VEL
LIN {X 0,Y 363.438,Z 362.888,A -85,B 0,C 180,E1 -13035.726,E2 -13035.726} C_VEL
LIN {X 0,Y 362.442,Z 372.606,A -85,B 0,C 180,E1 -13037.4,E2 -13037.4} C_VEL
LIN {X 0,Y 361.59,Z 380.347,A -85,B 0,C 180,E1 -13039.076,E2 -13039.076} C_VEL
LIN {X 0,Y 360.971,Z 387.497,A -85,B 0,C 180,E1 -13041.039,E2 -13041.039} C_VEL
LIN {X 0,Y 360.68,Z 392.264,A -85,B 0,C 180,E1 -13042.724,E2 -13042.724} C_VEL
LIN {X 0,Y 360.477,Z 395.908,A -85,B 0,C 180,E1 -13044.406,E2 -13044.406} C_VEL
LIN {X 0,Y 360.45,Z 397.792,A -85,B 0,C 180,E1 -13045.527,E2 -13045.527} C_VEL
LIN {X 0,Y 360.414,Z 400.213,A -85,B 0,C 180,E1 -13047.765,E2 -13047.765} C_VEL
LIN {X 0,Y 360.482,Z 400.833,A -85,B 0,C 180,E1 -13048.883,E2 -13048.883} C_VEL
LIN {X 0,Y 360.473,Z 401.051,A -85,B 0,C 180,E1 -13050,E2 -13050} C_VEL
LIN {X 0,Y 360.482,Z 400.832,A -85,B 0,C 180,E1 -13051.117,E2 -13051.117} C_VEL
LIN {X 0,Y 360.414,Z 400.212,A -85,B 0,C 180,E1 -13052.235,E2 -13052.235} C_VEL
LIN {X 0,Y 360.45,Z 397.789,A -85,B 0,C 180,E1 -13054.473,E2 -13054.473} C_VEL
LIN {X 0,Y 360.527,Z 394.76,A -85,B 0,C 180,E1 -13056.184,E2 -13056.184} C_VEL
LIN {X 0,Y 360.719,Z 390.801,A -85,B 0,C 180,E1 -13057.839,E2 -13057.839} C_VEL
LIN {X 0,Y 361.225,Z 384.639,A -85,B 0,C 180,E1 -13059.802,E2 -13059.802} C_VEL
LIN {X 0,Y 361.835,Z 377.912,A -85,B 0,C 180,E1 -13061.484,E2 -13061.484} C_VEL
LIN {X 0,Y 362.776,Z 369.583,A -85,B 0,C 180,E1 -13063.158,E2 -13063.158} C_VEL
LIN {X 0,Y 363.702,Z 361.05,A -85,B 0,C 180,E1 -13064.549,E2 -13064.549} C_VEL
LIN {X 0,Y 364.634,Z 350.505,A -85,B 0,C 180,E1 -13065.942,E2 -13065.942} C_VEL
LIN {X 0,Y 365.858,Z 338.663,A -85,B 0,C 180,E1 -13067.179,E2 -13067.179} C_VEL
LIN {X 0,Y 366.577,Z 329.25,A -85,B 0,C 180,E1 -13067.962,E2 -13067.962} C_VEL
LIN {X 0,Y 365.366,Z 318.094,A -85,B 0,C 180,E1 -13068.794,E2 -13068.794} C_VEL
LIN {X 0,Y 363.56,Z 304.967,A -85,B 0,C 180,E1 -13069.555,E2 -13069.555} C_VEL
LIN {X 0,Y 361.424,Z 293.054,A -85,B 0,C 180,E1 -13070.08,E2 -13070.08} C_VEL
LIN {X 0,Y 361.925,Z 286.046,A -85,B 0,C 180,E1 -13073.458,E2 -13073.458} C_VEL
LIN {X 0,Y 362.572,Z 278.808,A -85,B 0,C 180,E1 -13076.918,E2 -13076.918} C_VEL
LIN {X 0,Y 363.219,Z 272.003,A -85,B 0,C 180,E1 -13080.204,E2 -13080.204} C_VEL
LIN {X 0,Y 363.916,Z 265.642,A -85,B 0,C 180,E1 -13083.317,E2 -13083.317} C_VEL
LIN {X 0,Y 364.465,Z 260.54,A -85,B 0,C 180,E1 -13085.915,E2 -13085.915} C_VEL
LIN {X 0,Y 364.201,Z 256.468,A -85,B 0,C 180,E1 -13088.135,E2 -13088.135} C_VEL
LIN {X 0,Y 363.366,Z 251.356,A -85,B 0,C 180,E1 -13091.118,E2 -13091.118} C_VEL
LIN {X 0,Y 362.223,Z 245.181,A -85,B 0,C 180,E1 -13094.978,E2 -13094.978} C_VEL
LIN {X 0,Y 361.865,Z 243.412,A -85,B 0,C 180,E1 -13096.24,E2 -13096.24} C_VEL
LIN {X 0,Y 361.814,Z 243.414,A -85,B 0,C 180,E1 -13100.133,E2 -13100.133} C_VEL
LIN {X 0,Y 361.867,Z 243.409,A -85,B 0,C 180,E1 -13102.982,E2 -13102.982} C_VEL
LIN {X 0,Y 361.862,Z 243.412,A -85,B 0,C 180,E1 -13106.631,E2 -13106.631} C_VEL
LIN {X 0,Y 361.867,Z 243.406,A -85,B 0,C 180,E1 -13109.671,E2 -13109.671} C_VEL
LIN {X 0,Y 361.864,Z 243.407,A -85,B 0,C 180,E1 -13113.468,E2 -13113.468} C_VEL
LIN {X 0,Y 361.868,Z 243.406,A -85,B 0,C 180,E1 -13117.143,E2 -13117.143} C_VEL
LIN {X 0,Y 361.916,Z 243.401,A -85,B 0,C 180,E1 -13120.724,E2 -13120.724} C_VEL
LIN {X 0,Y 361.937,Z 243.397,A -85,B 0,C 180,E1 -13123.066,E2 -13123.066} C_VEL
LIN {X 0,Y 362.002,Z 243.39,A -85,B 0,C 180,E1 -13126.528,E2 -13126.528} C_VEL
LIN {X 0,Y 361.999,Z 243.394,A -85,B 0,C 180,E1 -13129.937,E2 -13129.937} C_VEL
LIN {X 0,Y 362.153,Z 243.373,A -85,B 0,C 180,E1 -13133.314,E2 -13133.314} C_VEL
LIN {X 0,Y 362.285,Z 243.358,A -85,B 0,C 180,E1 -13137.777,E2 -13137.777} C_VEL
LIN {X 0,Y 362.273,Z 243.356,A -85,B 0,C 180,E1 -13142.224,E2 -13142.224} C_VEL
LIN {X 0,Y 362.153,Z 243.371,A -85,B 0,C 180,E1 -13146.687,E2 -13146.687} C_VEL
LIN {X 0,Y 362.005,Z 243.389,A -85,B 0,C 180,E1 -13150.063,E2 -13150.063} C_VEL
LIN {X 0,Y 362.002,Z 243.389,A -85,B 0,C 180,E1 -13153.899,E2 -13153.899} C_VEL
LIN {X 0,Y 361.931,Z 243.404,A -85,B 0,C 180,E1 -13156.934,E2 -13156.934} C_VEL
LIN {X 0,Y 361.89,Z 243.406,A -85,B 0,C 180,E1 -13160.461,E2 -13160.461} C_VEL
LIN {X 0,Y 361.897,Z 243.403,A -85,B 0,C 180,E1 -13164.113,E2 -13164.113} C_VEL
LIN {X 0,Y 361.847,Z 243.409,A -85,B 0,C 180,E1 -13167.784,E2 -13167.784} C_VEL
LIN {X 0,Y 361.85,Z 243.408,A -85,B 0,C 180,E1 -13171.285,E2 -13171.285} C_VEL
LIN {X 0,Y 361.858,Z 243.412,A -85,B 0,C 180,E1 -13174.28,E2 -13174.28} C_VEL
LIN {X 0,Y 361.866,Z 243.406,A -85,B 0,C 180,E1 -13177.223,E2 -13177.223} C_VEL
LIN {X 0,Y 361.837,Z 243.411,A -85,B 0,C 180,E1 -13180.755,E2 -13180.755} C_VEL
LIN {X 0,Y 361.82,Z 243.415,A -85,B 0,C 180,E1 -13184.368,E2 -13184.368} C_VEL
LIN {X 0,Y 361.836,Z 243.412,A -85,B 0,C 180,E1 -13187.568,E2 -13187.568} C_VEL
LIN {X 0,Y 361.869,Z 243.406,A -85,B 0,C 180,E1 -13190.974,E2 -13190.974} C_VEL
LIN {X 0,Y 361.749,Z 243.422,A -85,B 0,C 180,E1 -13194.349,E2 -13194.349} C_VEL
LIN {X 0,Y 361.505,Z 243.456,A -85,B 0,C 180,E1 -13197.02,E2 -13197.02} C_VEL
LIN {X 0,Y 361.322,Z 243.618,A -85,B 0,C 180,E1 -13198.32,E2 -13198.32} C_VEL
LIN {X 0,Y 361.239,Z 246.972,A -85,B 0,C 180,E1 -13202.165,E2 -13202.165} C_VEL
LIN {X 0,Y 361.122,Z 250.4,A -85,B 0,C 180,E1 -13205.877,E2 -13205.877} C_VEL
LIN {X 0,Y 361.044,Z 254.528,A -85,B 0,C 180,E1 -13210.008,E2 -13210.008} C_VEL
LIN {X 0,Y 365.088,Z 268.582,A -85,B 0,C 180,E1 -13210.807,E2 -13210.807} C_VEL
LIN {X 0,Y 367.963,Z 281.087,A -85,B 0,C 180,E1 -13211.704,E2 -13211.704} C_VEL
LIN {X 0,Y 367.375,Z 292.846,A -85,B 0,C 180,E1 -13212.607,E2 -13212.607} C_VEL
LIN {X 0,Y 366.455,Z 303.553,A -85,B 0,C 180,E1 -13213.642,E2 -13213.642} C_VEL
LIN {X 0,Y 365.452,Z 314.355,A -85,B 0,C 180,E1 -13214.952,E2 -13214.952} C_VEL
LIN {X 0,Y 364.406,Z 323.499,A -85,B 0,C 180,E1 -13216.334,E2 -13216.334} C_VEL
LIN {X 0,Y 363.357,Z 332.371,A -85,B 0,C 180,E1 -13217.999,E2 -13217.999} C_VEL
LIN {X 0,Y 362.509,Z 339.508,A -85,B 0,C 180,E1 -13219.669,E2 -13219.669} C_VEL
LIN {X 0,Y 361.954,Z 344.318,A -85,B 0,C 180,E1 -13221.064,E2 -13221.064} C_VEL
LIN {X 0,Y 361.473,Z 348.539,A -85,B 0,C 180,E1 -13222.56,E2 -13222.56} C_VEL
LIN {X 0,Y 361.002,Z 352.565,A -85,B 0,C 180,E1 -13224.414,E2 -13224.414} C_VEL
LIN {X 0,Y 360.908,Z 354.405,A -85,B 0,C 180,E1 -13225.532,E2 -13225.532} C_VEL
LIN {X 0,Y 360.878,Z 355.787,A -85,B 0,C 180,E1 -13226.65,E2 -13226.65} C_VEL
LIN {X 0,Y 360.575,Z 357.392,A -85,B 0,C 180,E1 -13228.883,E2 -13228.883} C_VEL
LIN {X 0,Y 360.549,Z 357.624,A -85,B 0,C 180,E1 -13230,E2 -13230} C_VEL
LIN {X 0,Y 360.69,Z 356.85,A -85,B 0,C 180,E1 -13232.233,E2 -13232.233} C_VEL
LIN {X 0,Y 360.853,Z 355.886,A -85,B 0,C 180,E1 -13233.349,E2 -13233.349} C_VEL
LIN {X 0,Y 360.899,Z 354.545,A -85,B 0,C 180,E1 -13234.467,E2 -13234.467} C_VEL
LIN {X 0,Y 361.138,Z 351.702,A -85,B 0,C 180,E1 -13236.144,E2 -13236.144} C_VEL
LIN {X 0,Y 361.568,Z 347.839,A -85,B 0,C 180,E1 -13237.82,E2 -13237.82} C_VEL
LIN {X 0,Y 362.092,Z 342.857,A -85,B 0,C 180,E1 -13239.496,E2 -13239.496} C_VEL
LIN {X 0,Y 362.901,Z 336.572,A -85,B 0,C 180,E1 -13241.166,E2 -13241.166} C_VEL
LIN {X 0,Y 363.826,Z 328.705,A -85,B 0,C 180,E1 -13242.835,E2 -13242.835} C_VEL
LIN {X 0,Y 364.733,Z 320.681,A -85,B 0,C 180,E1 -13244.222,E2 -13244.222} C_VEL
LIN {X 0,Y 365.806,Z 310.879,A -85,B 0,C 180,E1 -13245.603,E2 -13245.603} C_VEL
LIN {X 0,Y 366.818,Z 299.848,A -85,B 0,C 180,E1 -13246.845,E2 -13246.845} C_VEL
LIN {X 0,Y 367.818,Z 287.87,A -85,B 0,C 180,E1 -13247.896,E2 -13247.896} C_VEL
LIN {X 0,Y 368.121,Z 281.613,A -85,B 0,C 180,E1 -13248.352,E2 -13248.352} C_VEL
LIN {X 0,Y 365.277,Z 269.344,A -85,B 0,C 180,E1 -13249.249,E2 -13249.249} C_VEL
LIN {X 0,Y 361.598,Z 256.626,A -85,B 0,C 180,E1 -13249.988,E2 -13249.988} C_VEL
LIN {X 0,Y 361.042,Z 254.466,A -85,B 0,C 180,E1 -13250.101,E2 -13250.101} C_VEL
LIN {X 0,Y 361.119,Z 250.509,A -85,B 0,C 180,E1 -13254.123,E2 -13254.123} C_VEL
LIN {X 0,Y 361.219,Z 247.077,A -85,B 0,C 180,E1 -13257.837,E2 -13257.837} C_VEL
LIN {X 0,Y 361.326,Z 243.716,A -85,B 0,C 180,E1 -13261.679,E2 -13261.679} C_VEL
LIN {X 0,Y 361.394,Z 243.584,A -85,B 0,C 180,E1 -13262.349,E2 -13262.349} C_VEL
LIN {X 0,Y 360.846,Z 243.551,A -85,B 0,C 180,E1 -13263.281,E2 -13263.281} C_VEL
LIN {X 0,Y 358.124,Z 243.874,A -85,B 0,C 180,E1 -13264.801,E2 -13264.801} C_VEL
LIN {X 0,Y 355.789,Z 244.167,A -85,B 0,C 180,E1 -13266.031,E2 -13266.031} C_VEL
LIN {X 0,Y 354.821,Z 244.285,A -85,B 0,C 180,E1 -13266.981,E2 -13266.981} C_VEL
LIN {X 0,Y 354.763,Z 244.292,A -85,B 0,C 180,E1 -13267.302,E2 -13267.302} C_VEL
LIN {X 0,Y 354.826,Z 244.284,A -85,B 0,C 180,E1 -13269.424,E2 -13269.424} C_VEL
LIN {X 0,Y 354.789,Z 244.288,A -85,B 0,C 180,E1 -13272.867,E2 -13272.867} C_VEL
LIN {X 0,Y 354.769,Z 244.295,A -85,B 0,C 180,E1 -13276.104,E2 -13276.104} C_VEL
LIN {X 0,Y 354.788,Z 244.289,A -85,B 0,C 180,E1 -13279.179,E2 -13279.179} C_VEL
LIN {X 0,Y 354.808,Z 244.286,A -85,B 0,C 180,E1 -13282.403,E2 -13282.403} C_VEL
LIN {X 0,Y 354.814,Z 244.285,A -85,B 0,C 180,E1 -13284.941,E2 -13284.941} C_VEL
LIN {X 0,Y 354.797,Z 244.287,A -85,B 0,C 180,E1 -13288.405,E2 -13288.405} C_VEL
LIN {X 0,Y 354.802,Z 244.291,A -85,B 0,C 180,E1 -13291.615,E2 -13291.615} C_VEL
LIN {X 0,Y 354.837,Z 244.285,A -85,B 0,C 180,E1 -13295.657,E2 -13295.657} C_VEL
LIN {X 0,Y 354.829,Z 244.287,A -85,B 0,C 180,E1 -13299.113,E2 -13299.113} C_VEL
LIN {X 0,Y 354.881,Z 244.278,A -85,B 0,C 180,E1 -13302.719,E2 -13302.719} C_VEL
LIN {X 0,Y 354.954,Z 244.267,A -85,B 0,C 180,E1 -13306.255,E2 -13306.255} C_VEL
LIN {X 0,Y 354.981,Z 244.264,A -85,B 0,C 180,E1 -13309.736,E2 -13309.736} C_VEL
LIN {X 0,Y 355.116,Z 244.247,A -85,B 0,C 180,E1 -13312.037,E2 -13312.037} C_VEL
LIN {X 0,Y 355.091,Z 244.252,A -85,B 0,C 180,E1 -13314.321,E2 -13314.321} C_VEL
LIN {X 0,Y 355.234,Z 244.232,A -85,B 0,C 180,E1 -13317.732,E2 -13317.732} C_VEL
LIN {X 0,Y 355.179,Z 244.24,A -85,B 0,C 180,E1 -13321.134,E2 -13321.134} C_VEL
LIN {X 0,Y 355.246,Z 244.235,A -85,B 0,C 180,E1 -13322.268,E2 -13322.268} C_VEL
LIN {X 0,Y 355.114,Z 244.249,A -85,B 0,C 180,E1 -13326.82,E2 -13326.82} C_VEL
LIN {X 0,Y 354.955,Z 244.273,A -85,B 0,C 180,E1 -13330.265,E2 -13330.265} C_VEL
LIN {X 0,Y 354.945,Z 244.273,A -85,B 0,C 180,E1 -13334.019,E2 -13334.019} C_VEL
LIN {X 0,Y 354.925,Z 244.276,A -85,B 0,C 180,E1 -13338.109,E2 -13338.109} C_VEL
LIN {X 0,Y 354.809,Z 244.289,A -85,B 0,C 180,E1 -13342.108,E2 -13342.108} C_VEL
LIN {X 0,Y 354.804,Z 244.292,A -85,B 0,C 180,E1 -13345.835,E2 -13345.835} C_VEL
LIN {X 0,Y 354.801,Z 244.293,A -85,B 0,C 180,E1 -13349.684,E2 -13349.684} C_VEL
LIN {X 0,Y 354.789,Z 244.289,A -85,B 0,C 180,E1 -13352.333,E2 -13352.333} C_VEL
LIN {X 0,Y 354.823,Z 244.287,A -85,B 0,C 180,E1 -13355.699,E2 -13355.699} C_VEL
LIN {X 0,Y 354.769,Z 244.295,A -85,B 0,C 180,E1 -13359.412,E2 -13359.412} C_VEL
LIN {X 0,Y 354.84,Z 244.417,A -85,B 0,C 180,E1 -13363.464,E2 -13363.464} C_VEL
LIN {X 0,Y 355.818,Z 249.719,A -85,B 0,C 180,E1 -13366.955,E2 -13366.955} C_VEL
LIN {X 0,Y 356.771,Z 255,A -85,B 0,C 180,E1 -13370.198,E2 -13370.198} C_VEL
LIN {X 0,Y 357.47,Z 260.133,A -85,B 0,C 180,E1 -13373.142,E2 -13373.142} C_VEL
LIN {X 0,Y 357.12,Z 265.019,A -85,B 0,C 180,E1 -13375.746,E2 -13375.746} C_VEL
LIN {X 0,Y 356.325,Z 271.711,A -85,B 0,C 180,E1 -13379.149,E2 -13379.149} C_VEL
LIN {X 0,Y 355.564,Z 279.063,A -85,B 0,C 180,E1 -13382.806,E2 -13382.806} C_VEL
LIN {X 0,Y 354.929,Z 285.827,A -85,B 0,C 180,E1 -13386.129,E2 -13386.129} C_VEL
LIN {X 0,Y 354.401,Z 292.703,A -85,B 0,C 180,E1 -13389.505,E2 -13389.505} C_VEL
LIN {X 0,Y 356.889,Z 306.536,A -85,B 0,C 180,E1 -13390.142,E2 -13390.142} C_VEL
LIN {X 0,Y 358.646,Z 319.794,A -85,B 0,C 180,E1 -13390.972,E2 -13390.972} C_VEL
